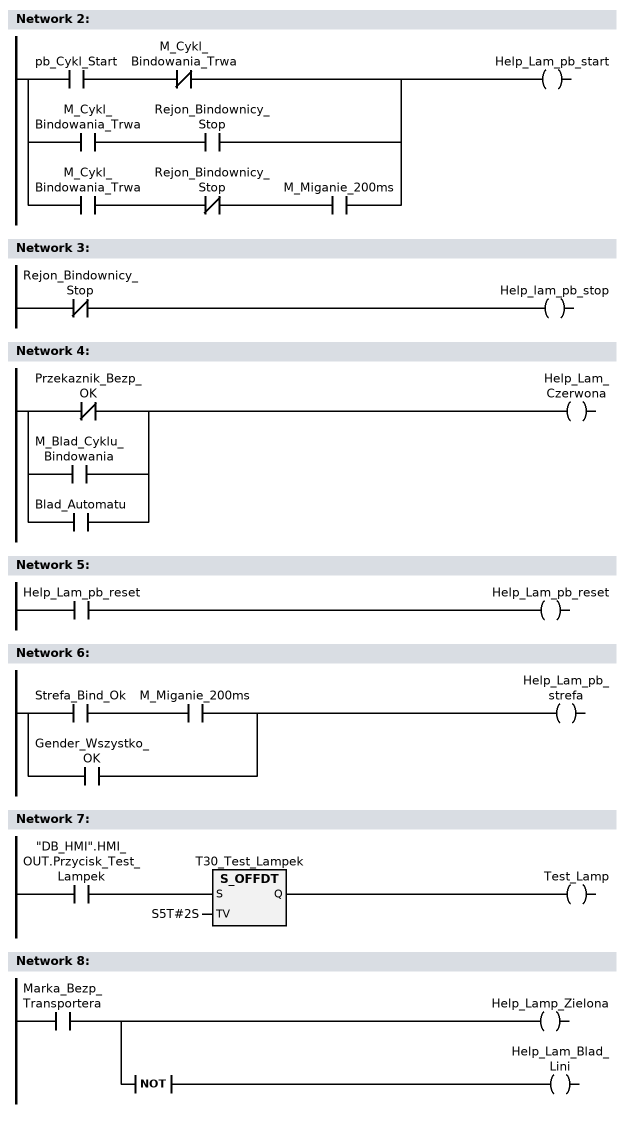
[picture p141: Sterwanie_Swiatlo networks 2-8]
NETWORK
TITLE =
//Lampka pb start cyklu
      A     "pb_Cykl_Start";
      AN    "M_Cykl_Bindowania_Trwa";
      O;
      A     "M_Cykl_Bindowania_Trwa";
      A     "Rejon_Bindownicy_Stop";
      O;
      A     "M_Cykl_Bindowania_Trwa";
      AN    "Rejon_Bindownicy_Stop";
      A     "M_Miganie_200ms";
      =     "Help_Lam_pb_start";
NETWORK
TITLE =
//Lampka stop
      AN    "Rejon_Bindownicy_Stop";
      =     "Help_lam_pb_stop";
NETWORK
TITLE =
      ON    "Przekaznik_Bezp_OK";
      O     "M_Blad_Cyklu_Bindowania";
      O     "Blad_Automatu";
      =     "Help_Lam_Czerwona";
NETWORK
TITLE =
//Miga reset
      A     "Help_Lam_pb_reset";
      =     "Help_Lam_pb_reset";
NETWORK
TITLE =
//Lampka bezpieczenstwa strefa
      A     "Strefa_Bind_Ok";
      A     "M_Miganie_200ms";
      O     "Gender_Wszystko_OK";
      =     "Help_Lam_pb_strefa";
NETWORK
TITLE =
//Test Lampek z timmerem przedluzonym
      A     "DB_HMI".HMI_OUT.Przycisk_Test_Lampek;
      L     S5T#2S;
      SF    "T30_Test_Lampek";
      NOP   0;
      NOP   0;
      NOP   0;
      A     "T30_Test_Lampek";
      =     "Test_Lamp";
NETWORK
TITLE =
//linia pracuje
      A     "Marka_Bezp_Transportera";
      =     L 1.0;
      A     L 1.0;
      BLD   102;
      =     "Help_Lamp_Zielona";
      A     L 1.0;
      NOT;
      =     "Help_Lam_Blad_Lini";
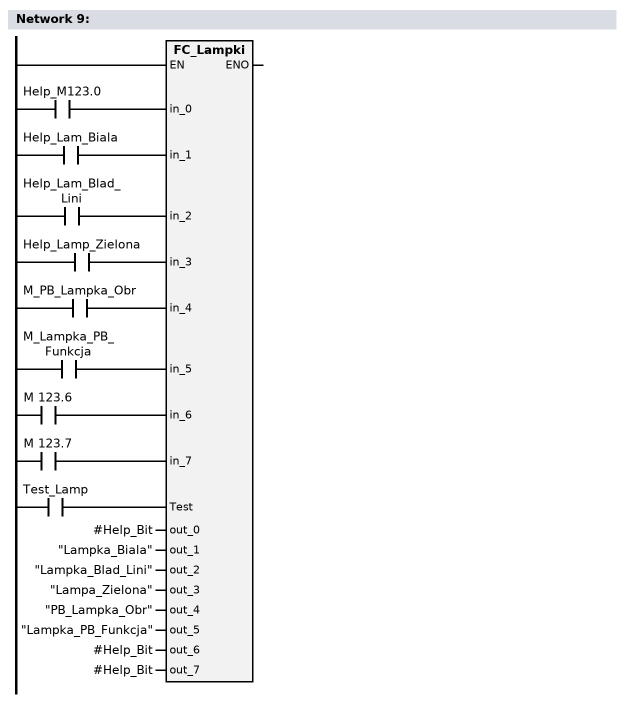
NETWORK
TITLE =
//Lampki na szafie sterowniczej sa troche przesuniete bo brakuje zielonej
      A     "Help_M123.0";
      =     L 1.0;
      BLD   103;
      A     "Help_Lam_Biala";
      =     L 1.1;
      BLD   103;
      A     "Help_Lam_Blad_Lini";
      =     L 1.2;
      BLD   103;
      A     "Help_Lamp_Zielona";
      =     L 1.3;
      BLD   103;
      A     "M_PB_Lampka_Obr";
      =     L 1.4;
      BLD   103;
      A     "M_Lampka_PB_Funkcja";
      =     L 1.5;
      BLD   103;
      A     M 123.6;
      =     L 1.6;
      BLD   103;
      A     M 123.7;
      =     L 1.7;
      BLD   103;
      A     "Test_Lamp";
      =     L 2.0;
      BLD   103;
      CALL  "FC_Lampki" (
           in_0                     := L 1.0,
           in_1                     := L 1.1,
           in_2                     := L 1.2,
           in_3                     := L 1.3,
           in_4                     := L 1.4,
           in_5                     := L 1.5,
           in_6                     := L 1.6,
           in_7                     := L 1.7,
           Test                     := L 2.0,
           out_0                    := #Help_Bit,
           out_1                    := "Lampka_Biala",
           out_2                    := "Lampka_Blad_Lini",
           out_3                    := "Lampa_Zielona",
           out_4                    := "PB_Lampka_Obr",
           out_5                    := "Lampka_PB_Funkcja",
           out_6                    := #Help_Bit,
           out_7                    := #Help_Bit);
      NOP   0;
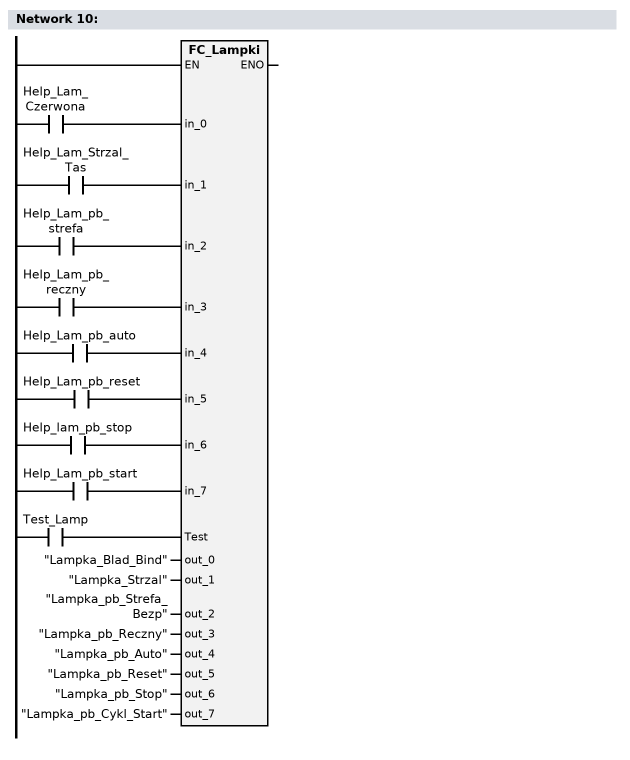
NETWORK
TITLE =
//funkcja zarzadzajaca lampami
//Lampki na panelu operatorskim
      A     "Help_Lam_Czerwona";
      =     L 1.0;
      BLD   103;
      A     "Help_Lam_Strzal_Tas";
      =     L 1.1;
      BLD   103;
      A     "Help_Lam_pb_strefa";
      =     L 1.2;
      BLD   103;
      A     "Help_Lam_pb_reczny";
      =     L 1.3;
      BLD   103;
      A     "Help_Lam_pb_auto";
      =     L 1.4;
      BLD   103;
      A     "Help_Lam_pb_reset";
      =     L 1.5;
      BLD   103;
      A     "Help_lam_pb_stop";
      =     L 1.6;
      BLD   103;
      A     "Help_Lam_pb_start";
      =     L 1.7;
      BLD   103;
      A     "Test_Lamp";
      =     L 2.0;
      BLD   103;
      CALL  "FC_Lampki" (
           in_0                     := L 1.0,
           in_1                     := L 1.1,
           in_2                     := L 1.2,
           in_3                     := L 1.3,
           in_4                     := L 1.4,
           in_5                     := L 1.5,
           in_6                     := L 1.6,
           in_7                     := L 1.7,
           Test                     := L 2.0,
           out_0                    := "Lampka_Blad_Bind",
           out_1                    := "Lampka_Strzal",
           out_2                    := "Lampka_pb_Strefa_Bezp",
           out_3                    := "Lampka_pb_Reczny",
           out_4                    := "Lampka_pb_Auto",
           out_5                    := "Lampka_pb_Reset",
           out_6                    := "Lampka_pb_Stop",
           out_7                    := "Lampka_pb_Cykl_Start");
      NOP   0;
END_FUNCTION

FUNCTION "Przyciski_Dwufunkcyjne" : VOID	// FC 11
AUTHOR : Kng
NAME : Help_FC
VERSION : 0.1
VAR_INPUT
  Kierunek_Prawo : BOOL ;
  Kierunek_Lewo : BOOL ;
  Funkcja : BOOL ;
END_VAR
VAR_OUTPUT
  Jazda_Prawo : BOOL ;
  Jazda_Lewo : BOOL ;
  Obrot_Prawo : BOOL ;
  Obrot_Lewo : BOOL ;
END_VAR
BEGIN
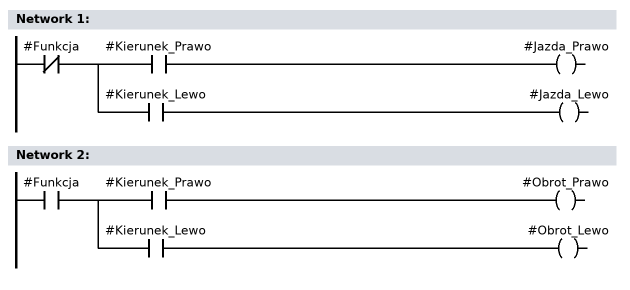
NETWORK
TITLE =
      AN    #Funkcja;
      =     L 0.0;
      A     L 0.0;
      A     #Kierunek_Prawo;
      =     #Jazda_Prawo;
      A     L 0.0;
      A     #Kierunek_Lewo;
      =     #Jazda_Lewo;
NETWORK
TITLE =
      A     #Funkcja;
      =     L 0.0;
      A     L 0.0;
      A     #Kierunek_Prawo;
      =     #Obrot_Prawo;
      A     L 0.0;
      A     #Kierunek_Lewo;
      =     #Obrot_Lewo;
END_FUNCTION

FUNCTION "Przyporzadkowanie_Wejsc" : VOID	// FC 20
//Pobranie z bloku db stanu wejsc sieci asi i przyporzadkowanie do odpowiedniego 
//urzadzenia lini.
//NW35-adresy B
//
//
//Opis sygnalow od bindownicy:
//banda 23, 24, 1, 2 tworza zestaw tasm maszyny bindujacej
//obr 15 to obrotnica bindownicy
//25,26- to kurtyny
//16-rygiel
//17-modul resetu
AUTHOR : Kng
NAME : Help_FC
VERSION : 0.1
VAR_TEMP
  Help_Bit_1 : BOOL ;
  Help_Bit_2 : BOOL ;
  Help_Word_1 : INT ;
  Help_Word_2 : INT ;
END_VAR
BEGIN
NETWORK
TITLE =
//Ten network celowo jest wolny
NETWORK
TITLE =
NETWORK
TITLE = Silnik ok
//Banda Adres 3
      A     "Asi_input_Transport".Adres_3_bit_0;
      =     "AIO".Banda_T3.Silnik_OK;
      A     "Asi_input_Transport".Adres_3_bit_1;
      =     "AIO".Banda_T3.Rezerwa_Silnik;
      A     "Asi_input_Transport".Adres_3_bit_2;
      =     "AIO".Banda_T3.Foto_1;
      A     "Asi_input_Transport".Adres_3_bit_3;
      =     "AIO".Banda_T3.Foto_2;
NETWORK
TITLE = Silnik ok
//Banda Adres 4
      A     "Asi_input_Transport".Adres_4_bit_0;
      =     "AIO".Banda_T4.Silnik_OK;
      A     "Asi_input_Transport".Adres_4_bit_1;
      =     "AIO".Banda_T4.Rezerwa_Silnik;
      A     "Asi_input_Transport".Adres_4_bit_2;
      =     "AIO".Banda_T4.Foto_1;
      A     "Asi_input_Transport".Adres_4_bit_3;
      =     "AIO".Banda_T4.Foto_2;
NETWORK
TITLE = Silnik ok
//Banda Adres 5
      A     "Asi_input_Transport".Adres_5_bit_0;
      =     "AIO".Banda_T5.Silnik_OK;
      A     "Asi_input_Transport".Adres_5_bit_1;
      =     "AIO".Banda_T5.Rezerwa_Silnik;
      A     "Asi_input_Transport".Adres_5_bit_2;
      =     "AIO".Banda_T5.Foto_1;
      A     "Asi_input_Transport".Adres_5_bit_3;
      =     "AIO".Banda_T5.Foto_2;
NETWORK
TITLE = Silnik ok
//Banda Adres 6
      A     "Asi_input_Transport".Adres_6_bit_0;
      =     "AIO".Banda_T6.Silnik_OK;
      A     "Asi_input_Transport".Adres_6_bit_1;
      =     "AIO".Banda_T6.Rezerwa_Silnik;
      A     "Asi_input_Transport".Adres_6_bit_2;
      =     "AIO".Banda_T6.Foto_1;
      A     "Asi_input_Transport".Adres_6_bit_3;
      =     "AIO".Banda_T6.Foto_2;
NETWORK
TITLE = Silnik ok
//Banda Adres 7
      A     "Asi_input_Transport".Adres_7_bit_0;
      =     "AIO".Banda_T7.Silnik_OK;
      A     "Asi_input_Transport".Adres_7_bit_1;
      =     "AIO".Banda_T7.Rezerwa_Silnik;
      A     "Asi_input_Transport".Adres_7_bit_2;
      =     "AIO".Banda_T7.Foto_1;
      A     "Asi_input_Transport".Adres_7_bit_3;
      =     "AIO".Banda_T7.Foto_2;
NETWORK
TITLE = Silnik ok
//Banda Adres 8
      A     "Asi_input_Transport".Adres_8_bit_0;
      =     "AIO".Banda_T8.Silnik_OK;
      A     "Asi_input_Transport".Adres_8_bit_1;
      =     "AIO".Banda_T8.Rezerwa_Silnik;
      A     "Asi_input_Transport".Adres_8_bit_2;
      =     "AIO".Banda_T8.Foto_1;
      A     "Asi_input_Transport".Adres_8_bit_3;
      =     "AIO".Banda_T8.Foto_2;
NETWORK
TITLE = Silnik ok
//Banda Adres 9
      A     "Asi_input_Transport".Adres_9_bit_0;
      =     "AIO".Banda_T9.Silnik_OK;
      A     "Asi_input_Transport".Adres_9_bit_1;
      =     "AIO".Banda_T9.Rezerwa_Silnik;
      A     "Asi_input_Transport".Adres_9_bit_2;
      =     "AIO".Banda_T9.Foto_1;
      A     "Asi_input_Transport".Adres_9_bit_3;
      =     "AIO".Banda_T9.Foto_2;
//Info do foliarki o zajetosci lini
      A     "AIO".Banda_T9.Foto_1;
      =     "MPI_GD".OUT.Foto_Banda_9;
//-
NETWORK
TITLE = Silnik ok
//Banda Adres 10.Banda nalezy do foliarki.
      A     "Asi_input_Transport".Adres_10_bit_0;
      =     "AIO".Banda_T10.Silnik_OK;
      A     "Asi_input_Transport".Adres_10_bit_1;
      =     "AIO".Banda_T10.Rezerwa_Silnik;
      A     "Asi_input_Transport".Adres_10_bit_2;
      =     "AIO".Banda_T10.Foto_1;
      A     "Asi_input_Transport".Adres_10_bit_3;
      =     "AIO".Banda_T10.Foto_2;
//Sygnaly do foliarki
      A     "AIO".Banda_T10.Silnik_OK;
      =     "MPI_GD".OUT.Silnik_10_OK;
//-
      A     "AIO".Banda_T10.Foto_1;
      =     "MPI_GD".OUT.Foto_1_Banda_10;
//-
      A     "AIO".Banda_T10.Foto_2;
      =     "MPI_GD".OUT.Foto_2_Banda_10;
NETWORK
TITLE = Silnik ok
//Banda Adres 11. Banda nalezy do foliarki.
      A     "Asi_input_Transport".Adres_11_bit_0;
      =     "AIO".Banda_T11.Silnik_OK;
      A     "Asi_input_Transport".Adres_11_bit_1;
      =     "AIO".Banda_T11.Rezerwa_Silnik;
      A     "Asi_input_Transport".Adres_11_bit_2;
      =     "AIO".Banda_T11.Foto_1;
      A     "Asi_input_Transport".Adres_11_bit_3;
      =     "AIO".Banda_T11.Foto_2;
//Sygnaly do foliarki
      A     "AIO".Banda_T11.Silnik_OK;
      =     "MPI_GD".OUT.Silnik_11_OK;
//-
      A     "AIO".Banda_T11.Foto_1;
      =     "MPI_GD".OUT.Foto_Banda_11;
NETWORK
TITLE = Silnik ok
//Banda Adres 12
      A     "Asi_input_Transport".Adres_12_bit_0;
      =     "AIO".Banda_T12.Silnik_OK;
      A     "Asi_input_Transport".Adres_12_bit_1;
      =     "AIO".Banda_T12.Rezerwa_Silnik;
      A     "Asi_input_Transport".Adres_12_bit_2;
      =     "AIO".Banda_T12.Foto_1;
      A     "Asi_input_Transport".Adres_12_bit_3;
      =     "AIO".Banda_T12.Foto_2;
NETWORK
TITLE = Silnik ok
//Banda Adres 13
      A     "Asi_input_Transport".Adres_13_bit_0;
      =     "AIO".Banda_T13.Silnik_OK;
      A     "Asi_input_Transport".Adres_13_bit_1;
      =     "AIO".Banda_T13.Rezerwa_Silnik;
      A     "Asi_input_Transport".Adres_13_bit_2;
      =     "AIO".Banda_T13.Foto_1;
      A     "Asi_input_Transport".Adres_13_bit_3;
      =     "AIO".Banda_T13.Foto_2;
NETWORK
TITLE = Silnik ok
//Banda Adres 14
      A     "Asi_input_Transport".Adres_14_bit_0;
      =     "AIO".Banda_T14.Silnik_OK;
      A     "Asi_input_Transport".Adres_14_bit_1;
      =     "AIO".Banda_T14.Rezerwa_Silnik;
      A     "Asi_input_Transport".Adres_14_bit_2;
      =     "AIO".Banda_T14.Foto_1;
      A     "Asi_input_Transport".Adres_14_bit_3;
      =     "AIO".Banda_T14.Foto_2;
NETWORK
TITLE = Silnik ok
//Obrotnica Adres_18 
      A     "Asi_input_Transport".Adres_18_bit_0;
      =     "AIO".Obr_T18.Silnik_OK;
      A     "Asi_input_Transport".Adres_18_bit_1;
      =     "AIO".Obr_T18.Rezerwa_Silnik;
      A     "Asi_input_Transport".Adres_18_bit_2;
      =     "AIO".Obr_T18.Foto_1;
      A     "Asi_input_Transport".Adres_18_bit_3;
      =     "AIO".Obr_T18.Foto_2;
NETWORK
TITLE = Silnik ok
//Czujniki obrotnicy 1 Adres 19
      A     "Asi_input_Transport".Adres_19_bit_0;
      =     "AIO".Czuj_T19.Czujnik_0_St;
      A     "Asi_input_Transport".Adres_19_bit_1;
      =     "AIO".Czuj_T19.Czujnik_Ham_0_St;
      A     "Asi_input_Transport".Adres_19_bit_2;
      =     "AIO".Czuj_T19.Czujnik_Ham_90_St;
      A     "Asi_input_Transport".Adres_19_bit_3;
      =     "AIO".Czuj_T19.Czujnik_90_St;
NETWORK
TITLE = Silnik ok
//Obrotnica Adres 20
      A     "Asi_input_Transport".Adres_20_bit_0;
      =     "AIO".Obr_T20.Silnik_OK;
      A     "Asi_input_Transport".Adres_20_bit_1;
      =     "AIO".Obr_T20.Rezerwa_Silnik;
      A     "Asi_input_Transport".Adres_20_bit_2;
      =     "AIO".Obr_T20.Foto_1;
      A     "Asi_input_Transport".Adres_20_bit_3;
      =     "AIO".Obr_T20.Foto_2;
NETWORK
TITLE = Silnik ok
//Czujniki Obrotnicy 2 Adres 21
      A     "Asi_input_Transport".Adres_21_bit_0;
      =     "AIO".Czuj_T21.Czujnik_0_St;
      A     "Asi_input_Transport".Adres_21_bit_1;
      =     "AIO".Czuj_T21.Czujnik_Ham_0_St;
      A     "Asi_input_Transport".Adres_21_bit_2;
      =     "AIO".Czuj_T21.Czujnik_Ham_90_St;
      A     "Asi_input_Transport".Adres_21_bit_3;
      =     "AIO".Czuj_T21.Czujnik_90_St;
NETWORK
TITLE = Silnik ok
//Czujniki Obrotnicy 2 Adres 22
      A     "Asi_input_Transport".Adres_22_bit_0;
      =     "AIO".Czuj_T22.Czujnik_45_St_CW;
      A     "Asi_input_Transport".Adres_22_bit_1;
      =     "AIO".Czuj_T22.Czujnik_45_St_CCW;
      A     "Asi_input_Transport".Adres_22_bit_2;
      =     "AIO".Czuj_T22.Rez_0_2;
      A     "Asi_input_Transport".Adres_22_bit_3;
      =     "AIO".Czuj_T22.Rez_0_3;
NETWORK
TITLE = Silnik ok
//Sprawdzenie czujnikow Bezpieczenstwa lini
//Not Aus 27 
      A     "Asi_input_Transport".Adres_27_bit_0;
      =     "AIO".ESTOP_T27.EStop_Tor_1_1;
      A     "Asi_input_Transport".Adres_27_bit_1;
      =     "AIO".ESTOP_T27.EStop_Tor_1_2;
      A     "Asi_input_Transport".Adres_27_bit_2;
      =     "AIO".ESTOP_T27.EStop_Tor_2_1;
      A     "Asi_input_Transport".Adres_27_bit_3;
      =     "AIO".ESTOP_T27.EStop_Tor_2_2;
NETWORK
TITLE =
//Sprawdzenie czujnikow Bezpieczenstwa lini
//Not Aus 28
      A     "Asi_input_Transport".Adres_28_bit_0;
      =     "AIO".ESTOP_T28.EStop_Tor_1_1;
      A     "Asi_input_Transport".Adres_28_bit_1;
      =     "AIO".ESTOP_T28.EStop_Tor_1_2;
      A     "Asi_input_Transport".Adres_28_bit_2;
      =     "AIO".ESTOP_T28.EStop_Tor_2_1;
      A     "Asi_input_Transport".Adres_28_bit_3;
      =     "AIO".ESTOP_T28.EStop_Tor_2_2;
NETWORK
TITLE =
//Sprawdzenie czujnikow Bezpieczenstwa lini
//Not Aus 29
      A     "Asi_input_Transport".Adres_29_bit_0;
      =     "AIO".ESTOP_T29.EStop_Tor_1_1;
      A     "Asi_input_Transport".Adres_29_bit_1;
      =     "AIO".ESTOP_T29.EStop_Tor_1_2;
      A     "Asi_input_Transport".Adres_29_bit_2;
      =     "AIO".ESTOP_T29.EStop_Tor_2_1;
      A     "Asi_input_Transport".Adres_29_bit_3;
      =     "AIO".ESTOP_T29.EStop_Tor_2_2;
NETWORK
TITLE =
//Sprawdzenie czujnikow Bezpieczenstwa lini
//Not Aus 30
      A     "Asi_input_Transport".Adres_30_bit_0;
      =     "AIO".ESTOP_T30.EStop_Tor_1_1;
      A     "Asi_input_Transport".Adres_30_bit_1;
      =     "AIO".ESTOP_T30.EStop_Tor_1_2;
      A     "Asi_input_Transport".Adres_30_bit_2;
      =     "AIO".ESTOP_T30.EStop_Tor_2_1;
      A     "Asi_input_Transport".Adres_30_bit_3;
      =     "AIO".ESTOP_T30.EStop_Tor_2_2;
END_FUNCTION

FUNCTION "Przyporzadkowanie_Wyjsc" : VOID	// FC 21
VERSION : 0.1
VAR_TEMP
  Temp_Word_1 : INT ;
  Help_Bit_1 : BOOL ;
END_VAR
BEGIN
NETWORK
TITLE =
//Ten Network celowo jest wolny
NETWORK
TITLE = Temporary placeholder variable
//Banda 3 Adres 3
//****************ClockWise*******************
      A     "Zawsze_False";	//C_Wise
      =     "Asi_output_Transport".Adres_3_bit_0;
//****************CounterClockWise************
      A     "AIO".Banda_T3.C_Wise;
      =     "Asi_output_Transport".Adres_3_bit_1;	//CC_Wise
//****************Wolno***********************
      A     "Zawsze_True";
      =     "Asi_output_Transport".Adres_3_bit_2;	//Wolno
//****************Bit_Bezpieczenstwa**********
      A     "Marka_Bezp_Transportera";	//Safety
      =     "Asi_output_Transport".Adres_3_bit_3;
NETWORK
TITLE = Temporary placeholder variable
//Banda 4 Obrotnica
//****************ClockWise*******************
      A     "AIO".Banda_T4.C_Wise;	//C_Wise
      =     "Asi_output_Transport".Adres_4_bit_0;
//****************CounterClockWise************
      A     "AIO".Banda_T4.CC_Wise;
      =     "Asi_output_Transport".Adres_4_bit_1;	//CC_Wise
//****************Wolno***********************
      A     "Zawsze_True";
      =     "Asi_output_Transport".Adres_4_bit_2;	//Wolno
//****************Bit_Bezpieczenstwa**********
      A     "Marka_Bezp_Transportera";	//Safety
      =     "Asi_output_Transport".Adres_4_bit_3;
NETWORK
TITLE = Temporary placeholder variable
//Banda 5 Rolki
//****************ClockWise*******************
      A     "Zawsze_False";	//C_Wise
      =     "Asi_output_Transport".Adres_5_bit_0;
//****************CounterClockWise************
      A     "AIO".Banda_T5.C_Wise;
      =     "Asi_output_Transport".Adres_5_bit_1;	//CC_Wise
//****************Wolno***********************
      A     "Zawsze_True";
      =     "Asi_output_Transport".Adres_5_bit_2;	//Wolno
//****************Bit_Bezpieczenstwa**********
      A     "Marka_Bezp_Transportera";	//Safety
      =     "Asi_output_Transport".Adres_5_bit_3;
NETWORK
TITLE = Temporary placeholder variable
//Banda 6 Rolki
//****************ClockWise*******************
      A     "AIO".Banda_T6.C_Wise;	//C_Wise
      =     "Asi_output_Transport".Adres_6_bit_0;
//****************CounterClockWise************
      A     "Zawsze_False";
      =     "Asi_output_Transport".Adres_6_bit_1;	//CC_Wise
//****************Wolno***********************
      A     "Zawsze_False";
      =     "Asi_output_Transport".Adres_6_bit_2;	//Wolno
//****************Bit_Bezpieczenstwa**********
      A     "Marka_Bezp_Transportera";	//Safety
      =     "Asi_output_Transport".Adres_6_bit_3;
NETWORK
TITLE = Temporary placeholder variable
//Banda 7 Rolki
//****************ClockWise*******************
      A     "Zawsze_False";	//C_Wise
      =     "Asi_output_Transport".Adres_7_bit_0;
//****************CounterClockWise************
      A     "AIO".Banda_T7.C_Wise;
      =     "Asi_output_Transport".Adres_7_bit_1;	//CC_Wise
//****************Wolno***********************
      A     "Zawsze_True";
      =     "Asi_output_Transport".Adres_7_bit_2;	//Wolno
//****************Bit_Bezpieczenstwa**********
      A     "Marka_Bezp_Transportera";	//Safety
      =     "Asi_output_Transport".Adres_7_bit_3;
NETWORK
TITLE = Temporary placeholder variable
//Banda 8 Rolki
//****************ClockWise*******************
      A     "AIO".Banda_T8.C_Wise;	//C_Wise
      =     "Asi_output_Transport".Adres_8_bit_0;
//****************CounterClockWise************
      A     "Zawsze_False";
      =     "Asi_output_Transport".Adres_8_bit_1;	//CC_Wise
//****************Wolno***********************
      A     "Zawsze_False";
      =     "Asi_output_Transport".Adres_8_bit_2;	//Wolno
//****************Bit_Bezpieczenstwa**********
      A     "Marka_Bezp_Transportera";	//Safety
      =     "Asi_output_Transport".Adres_8_bit_3;
NETWORK
TITLE = Temporary placeholder variable
//Banda 9 Rolki
//****************ClockWise*******************
      A     "Zawsze_False";	//C_Wise
      =     "Asi_output_Transport".Adres_9_bit_0;
//****************CounterClockWise************
      A     "AIO".Banda_T9.C_Wise;
      =     "Asi_output_Transport".Adres_9_bit_1;	//CC_Wise
//****************Wolno***********************
      A     "Zawsze_True";
      =     "Asi_output_Transport".Adres_9_bit_2;	//Wolno
//****************Bit_Bezpieczenstwa**********
      A     "Marka_Bezp_Transportera";	//Safety
      =     "Asi_output_Transport".Adres_9_bit_3;
NETWORK
TITLE = Temporary placeholder variable
//Banda 10 Rolki
//Uwaga Banda ta nalezy do foliarki
//Sygnaly z foliarki
      A     "MPI_GD".IN.Motor_10_Lewo;
      =     "AIO".Banda_T10.C_Wise;
      A     "MPI_GD".IN.Motor_10_Prawo;
      =     "AIO".Banda_T10.CC_Wise;
//****************ClockWise*******************
      A     "AIO".Banda_T10.C_Wise;	//C_Wise
      =     "Asi_output_Transport".Adres_10_bit_0;
//****************CounterClockWise************
      A     "AIO".Banda_T10.CC_Wise;
      =     "Asi_output_Transport".Adres_10_bit_1;	//CC_Wise
//****************Wolno***********************
      A     "Zawsze_True";
      =     "Asi_output_Transport".Adres_10_bit_2;	//Wolno
//****************Bit_Bezpieczenstwa**********
      A     "Marka_Bezp_Transportera";	//Safety
      =     "Asi_output_Transport".Adres_10_bit_3;
NETWORK
TITLE = Temporary placeholder variable
//Banda 11 Rolki
//Uwaga Banda ta nalezy do foliarki
//Sygnaly z foliarki
      A     "MPI_GD".IN.Motor_11_Lewo;
      =     "AIO".Banda_T11.C_Wise;
      A     "MPI_GD".IN.Motor_11_Prawo;
      =     "AIO".Banda_T11.CC_Wise;
//****************ClockWise*******************
      A     "AIO".Banda_T11.C_Wise;	//C_Wise
      =     "Asi_output_Transport".Adres_11_bit_0;
//****************CounterClockWise************
      A     "AIO".Banda_T11.CC_Wise;
      =     "Asi_output_Transport".Adres_11_bit_1;	//CC_Wise
//****************Wolno***********************
      A     "Zawsze_True";
      =     "Asi_output_Transport".Adres_11_bit_2;	//Wolno
//****************Bit_Bezpieczenstwa**********
      A     "Marka_Bezp_Transportera";	//Safety
      =     "Asi_output_Transport".Adres_11_bit_3;
NETWORK
TITLE = Temporary placeholder variable
//Banda 12 Rolki wlot 2 na obrotnice
//****************ClockWise*******************
      A     "AIO".Banda_T12.C_Wise;	//C_Wise
      =     "Asi_output_Transport".Adres_12_bit_0;
//****************CounterClockWise************
      A     "Zawsze_False";
      =     "Asi_output_Transport".Adres_12_bit_1;	//CC_Wise
//****************Wolno***********************
      A     "Zawsze_False";
      =     "Asi_output_Transport".Adres_12_bit_2;	//Wolno
//****************Bit_Bezpieczenstwa**********
      A     "Marka_Bezp_Transportera";	//Safety
      =     "Asi_output_Transport".Adres_12_bit_3;
NETWORK
TITLE = Temporary placeholder variable
//Banda 13 Adres 13 Rolki na obrotnicy
//****************ClockWise*******************
      A     "AIO".Banda_T13.C_Wise;	//C_Wise
      =     "Asi_output_Transport".Adres_13_bit_0;
//****************CounterClockWise************
      A     "AIO".Banda_T13.CC_Wise;
      =     "Asi_output_Transport".Adres_13_bit_1;	//CC_Wise
//****************Wolno***********************
      A     "Zawsze_False";
      =     "Asi_output_Transport".Adres_13_bit_2;	//Wolno
//****************Bit_Bezpieczenstwa**********
      A     "Marka_Bezp_Transportera";	//Safety
      =     "Asi_output_Transport".Adres_13_bit_3;
NETWORK
TITLE = Temporary placeholder variable
//Banda 14 Adres 14 Wylot z maszyny
//****************ClockWise*******************
      A     "AIO".Banda_T14.C_Wise;	//C_Wise
      =     "Asi_output_Transport".Adres_14_bit_0;
//****************CounterClockWise************
      A     "Zawsze_False";
      =     "Asi_output_Transport".Adres_14_bit_1;	//CC_Wise
//****************Wolno***********************
      A     "Zawsze_False";
      =     "Asi_output_Transport".Adres_14_bit_2;	//Wolno
//****************Bit_Bezpieczenstwa**********
      A     "Marka_Bezp_Transportera";	//Safety
      =     "Asi_output_Transport".Adres_14_bit_3;
NETWORK
TITLE = Temporary placeholder variable
//Obrotnica 18  Adres 18 
//****************ClockWise*******************
      A     "AIO".Obr_T18.C_Wise;
      =     "Asi_output_Transport".Adres_18_bit_0;
//****************CounterClockWise************
      A     "AIO".Obr_T18.CC_Wise;
      =     "Asi_output_Transport".Adres_18_bit_1;	//CC_Wise
//****************Wolno***********************
      A     "AIO".Obr_T18.Wolno;
      =     "Asi_output_Transport".Adres_18_bit_2;	//Wolno
//****************Bit_Bezpieczenstwa**********
      A     "Marka_Bezp_Transportera";	//Safety
      =     "Asi_output_Transport".Adres_18_bit_3;
NETWORK
TITLE = Temporary placeholder variable
//Obrotnica 20 Adres 20
//****************ClockWise*******************
      A     "AIO".Obr_T20.C_Wise;
      =     "Asi_output_Transport".Adres_20_bit_0;
//****************CounterClockWise************
      A     "AIO".Obr_T20.CC_Wise;
      =     "Asi_output_Transport".Adres_20_bit_1;	//CC_Wise
//****************Wolno***********************
      A     "AIO".Obr_T20.Wolno;
      =     "Asi_output_Transport".Adres_20_bit_2;	//Wolno
//****************Bit_Bezpieczenstwa**********
      A     "Marka_Bezp_Transportera";	//Safety
      =     "Asi_output_Transport".Adres_20_bit_3;
NETWORK
TITLE = Temporary placeholder variable
//Adres 21, 22 Brak Output
NETWORK
TITLE =
//Aedrs 27,28,29,30,31. Adresy ESTOP brak syganlow output
NETWORK
TITLE =
//Dziekuje za uwage
END_FUNCTION

FUNCTION "Przyp_Wejsc_Gender" : VOID	// FC 22
//Pobranie z bloku db stanu wejsc sieci asi i przyporzadkowanie do odpowiedniego 
//urzadzenia lini.
//NW35-adresy B
//
//
//Opis sygnalow od bindownicy:
//banda 23, 24, 1, 2 tworza zestaw tasm maszyny bindujacej
//obr 15 to obrotnica bindownicy
//25,26- to kurtyny
//16-rygiel
//17-modul resetu
AUTHOR : Kng
NAME : Help_FC
VERSION : 0.1
VAR_TEMP
  Help_Bit_1 : BOOL ;
  Help_Bit_2 : BOOL ;
  Help_Word_1 : INT ;
  Help_Word_2 : INT ;
END_VAR
BEGIN
NETWORK
TITLE =
//Ten network celowo jest wolny
NETWORK
TITLE =
NETWORK
TITLE = Silnik ok
//Banda Adres 1 (nowy) rolki obrotnica
      A     "Asi_Input_Gender".Adres_1_bit_0;
      O     "Zawsze_True";	//dodane
      =     "AIO".Banda_G1.Silnik_OK;
      A     "Asi_Input_Gender".Adres_1_bit_1;
      =     "AIO".Banda_G1.Rezerwa_Silnik;
      A     "Asi_Input_Gender".Adres_1_bit_2;
      =     "AIO".Banda_G1.Foto_1;
      A     "Asi_Input_Gender".Adres_1_bit_3;
      =     "AIO".Banda_G1.Foto_2;
NETWORK
TITLE = Silnik ok
//Banda Adres 2 (nowy)
      A     "Asi_Input_Gender".Adres_2_bit_0;
      O     "Zawsze_True";
      =     "AIO".Banda_G2.Silnik_OK;
      A     "Asi_Input_Gender".Adres_2_bit_1;
      =     "AIO".Banda_G2.Rezerwa_Silnik;
      A     "Asi_Input_Gender".Adres_2_bit_2;
      =     "AIO".Banda_G2.Foto_1;
      A     "Asi_Input_Gender".Adres_2_bit_3;
      =     "AIO".Banda_G2.Foto_2;
NETWORK
TITLE = Silnik ok
//Obrotnica Adres 15 (nowy)
      A     "Asi_Input_Gender".Adres_15_bit_0;
      =     "AIO".Obr_G15.Silnik_OK;
      A     "Asi_Input_Gender".Adres_15_bit_1;
      =     "AIO".Obr_G15.Rezerwa_Silnik;
      A     "Asi_Input_Gender".Adres_15_bit_2;
      =     "AIO".Obr_G15.Foto_1;
      A     "Asi_Input_Gender".Adres_15_bit_3;
      =     "AIO".Obr_G15.Foto_2;
NETWORK
TITLE = Silnik ok
//Uwaga modul safety !!! (nowy)
//Rygiel Adres 16
      A     "Asi_Input_Gender".Adres_16_bit_0;
      =     "AIO".Rygiel_TG16.OSSD_Tor_1_1;
      A     "Asi_Input_Gender".Adres_16_bit_1;
      =     "AIO".Rygiel_TG16.OSSD_Tor_1_2;
      A     "Asi_Input_Gender".Adres_16_bit_2;
      =     "AIO".Rygiel_TG16.OSSD_Tor_2_1;
      A     "Asi_Input_Gender".Adres_16_bit_3;
      =     "AIO".Rygiel_TG16.OSSD_Tor_2_2;
NETWORK
TITLE = Silnik ok
//Reset kurtyn bezpieczenswa Adres 17 (nowy)
//Nie wykorzystywane wejscia
NETWORK
TITLE = Wejscie SEW 1
//Banda 23 znajdujaca sie bedaca banda wjazdowa do bindownicy (nowy)
      A     "Asi_Input_Gender".Adres_23_bit_0;
      =     "AIO".Banda_G23.Silnik_OK;
      A     "Asi_Input_Gender".Adres_23_bit_1;
      =     "AIO".Banda_G23.Rezerwa_Silnik;
      A     "Asi_Input_Gender".Adres_23_bit_2;
      =     "AIO".Banda_G23.Foto_1;
      A     "Asi_Input_Gender".Adres_23_bit_3;
      =     "AIO".Banda_G23.Foto_2;
NETWORK
TITLE = Silnik ok
//Banda 24 (nowy)
      A     "Asi_Input_Gender".Adres_24_bit_0;
      =     "AIO".Banda_G24.Silnik_OK;
      A     "Asi_Input_Gender".Adres_24_bit_1;
      =     "AIO".Banda_G24.Rezerwa_Silnik;
      A     "Asi_Input_Gender".Adres_24_bit_2;
      =     "AIO".Banda_G24.Foto_1;
      A     "Asi_Input_Gender".Adres_24_bit_3;
      =     "AIO".Banda_G24.Foto_2;
NETWORK
TITLE =
//Sprawdzenie czujnikow Bezpieczenstwa lini
//Kurtyna 25 (nowy)
      A     "Asi_Input_Gender".Adres_25_bit_0;
      =     "AIO".Kurtyna_G25.OSSD_Tor_1_1;
      A     "Asi_Input_Gender".Adres_25_bit_1;
      =     "AIO".Kurtyna_G25.OSSD_Tor_1_2;
      A     "Asi_Input_Gender".Adres_25_bit_2;
      =     "AIO".Kurtyna_G25.OSSD_Tor_2_1;
      A     "Asi_Input_Gender".Adres_25_bit_3;
      =     "AIO".Kurtyna_G25.OSSD_Tor_2_2;
NETWORK
TITLE =
//Sprawdzenie czujnikow Bezpieczenstwa lini
//Kurtyna 26 (nowy)
      A     "Asi_Input_Gender".Adres_26_bit_0;
      =     "AIO".Kurtyna_G26.OSSD_Tor_1_1;
      A     "Asi_Input_Gender".Adres_26_bit_1;
      =     "AIO".Kurtyna_G26.OSSD_Tor_1_2;
      A     "Asi_Input_Gender".Adres_26_bit_2;
      =     "AIO".Kurtyna_G26.OSSD_Tor_2_1;
      A     "Asi_Input_Gender".Adres_26_bit_3;
      =     "AIO".Kurtyna_G26.OSSD_Tor_2_2;
NETWORK
TITLE =
//Sprawdzenie czujnikow Bezpieczenstwa lini
//Not Aus 31 (nowy)
      A     "Asi_Input_Gender".Adres_31_bit_0;
      =     "AIO".ESTOP_TG31.EStop_Tor_1_1;
      A     "Asi_Input_Gender".Adres_31_bit_1;
      =     "AIO".ESTOP_TG31.EStop_Tor_1_2;
      A     "Asi_Input_Gender".Adres_31_bit_2;
      =     "AIO".ESTOP_TG31.EStop_Tor_2_1;
      A     "Asi_Input_Gender".Adres_31_bit_3;
      =     "AIO".ESTOP_TG31.EStop_Tor_2_2;
NETWORK
TITLE =
//Segment adresow B
//Dotyczy jedynie bialych modulow inuput nie zawartych wyzej
NETWORK
TITLE =
//Czujnik bindownicy Adres 19B (nowy)
      A     "Asi_Input_Gender".B_Adres_19_bit_0;
      =     "AIO".Czuj_G19_B.Czujnik_0_St;
      A     "Asi_Input_Gender".B_Adres_19_bit_1;
      =     "AIO".Czuj_G19_B.Czujnik_Ham_0_St;
      A     "Asi_Input_Gender".B_Adres_19_bit_2;
      =     "AIO".Czuj_G19_B.Czujnik_Ham_90_St;
      A     "Asi_Input_Gender".B_Adres_19_bit_3;
      =     "AIO".Czuj_G19_B.Czujnik_90_St;
NETWORK
TITLE =
//Czujnik bindownicy Adres 17B (nowy)
      A     "Asi_Input_Gender".B_Adres_17_bit_0;
      =     "AIO".Czuj_G17_B.Czujnik_Ham_180_St;
      A     "Asi_Input_Gender".B_Adres_17_bit_1;
      =     "AIO".Czuj_G17_B.Czujnik_180_St;
      A     "Asi_Input_Gender".B_Adres_17_bit_2;
      =     "AIO".Czuj_G17_B.Czujnik_Ham_270_St;
      A     "Asi_Input_Gender".B_Adres_17_bit_3;
      =     "AIO".Czuj_G17_B.Czujnik_270_St;
END_FUNCTION

FUNCTION "Przyp_Wysc_Gender" : VOID	// FC 23
VERSION : 0.1
VAR_TEMP
  Temp_Word_1 : INT ;
  Help_Bit_1 : BOOL ;
END_VAR
BEGIN
NETWORK
TITLE =
//Ten Network celowo jest wolny
NETWORK
TITLE = Temporary placeholder variable
//Banda 1 Adres 1 (nowy)
//****************ClockWise*******************
      A     "AIO".Banda_G1.CC_Wise;	//C_Wise
      =     "Asi_Output_Gender".Adres_1_bit_0;
//****************CounterClockWise************
      A     "AIO".Banda_G1.C_Wise;
      =     "Asi_Output_Gender".Adres_1_bit_1;	//CC_Wise
//****************Wolno***********************
      A     "AIO".Banda_G1.Wolno;
      O     "pb_Strefa_bezpieczenstwa";
      =     "Asi_Output_Gender".Adres_1_bit_2;	//Wolno
//****************Bit_Bezpieczenstwa**********
      A     "Marka_Bezp_Gendera";	//Safety
      =     "Asi_Output_Gender".Adres_1_bit_3;
NETWORK
TITLE = Temporary placeholder variable
//Banda 2 Adres 2 (nowy)
//****************ClockWise*******************
      A     "AIO".Banda_G2.CC_Wise;	//C_Wise
      =     "Asi_Output_Gender".Adres_2_bit_0;
//****************CounterClockWise************
      A     "AIO".Banda_G2.C_Wise;
      =     "Asi_Output_Gender".Adres_2_bit_1;	//CC_Wise
//****************Wolno***********************
      AN    "AIO".Banda_G2.Wolno;
      =     "Asi_Output_Gender".Adres_2_bit_2;	//Wolno
//****************Bit_Bezpieczenstwa**********
      A     "Marka_Bezp_Gendera";	//Safety
      =     "Asi_Output_Gender".Adres_2_bit_3;
NETWORK
TITLE = Temporary placeholder variable
//Obrotnica 15 Adres 15 (nowy)
//****************ClockWise*******************
      A     "AIO".Obr_G15.C_Wise;
      =     "Asi_Output_Gender".Adres_15_bit_0;
//****************CounterClockWise************
      A     "AIO".Obr_G15.CC_Wise;
      =     "Asi_Output_Gender".Adres_15_bit_1;	//CC_Wise
//****************Wolno***********************
      AN    "AIO".Obr_G15.Wolno;
      =     "Asi_Output_Gender".Adres_15_bit_2;	//Wolno
//****************Bit_Bezpieczenstwa**********
      A     "Marka_Bezp_Gendera";	//Safety
      =     "Asi_Output_Gender".Adres_15_bit_3;
NETWORK
TITLE =
//adres 16 rygiel brak output (nowy)
NETWORK
TITLE = Temporary placeholder variable
//adres 17 reset kurtyn (nowy)
//****************Reset wlot *****************
      A     "AIO".Reset_TG17.Reset_Wlot;
      =     "Asi_Output_Gender".Adres_17_bit_0;	//reset wlot
//****************Reset wylot ****************
      A     "AIO".Reset_TG17.Reset_Wylot;
      =     "Asi_Output_Gender".Adres_17_bit_1;	//reset wylot
NETWORK
TITLE = Temporary placeholder variable
//Banda 23 (nowy)
//
//****************ClockWise*******************
      A     "AIO".Banda_G23.CC_Wise;	//C_Wise
      =     "Asi_Output_Gender".Adres_23_bit_0;
//****************CounterClockWise************
      A     "AIO".Banda_G23.C_Wise;
      =     "Asi_Output_Gender".Adres_23_bit_1;	//CC_Wise
//****************Wolno***********************
      A     "AIO".Banda_G23.Wolno;
      =     "Asi_Output_Gender".Adres_23_bit_2;	//Wolno
//****************Bit_Bezpieczenstwa**********
      A     "Marka_Bezp_Gendera";	//Safety
      =     "Asi_Output_Gender".Adres_23_bit_3;
NETWORK
TITLE = Temporary placeholder variable
//Banda 24 (nowy)
//
//****************ClockWise*******************
      A     "AIO".Banda_G24.CC_Wise;	//C_Wise
      =     "Asi_Output_Gender".Adres_24_bit_0;
//****************CounterClockWise************
      A     "AIO".Banda_G24.C_Wise;
      =     "Asi_Output_Gender".Adres_24_bit_1;	//CC_Wise
//****************Wolno***********************
      A     "Zawsze_True";
      =     "Asi_Output_Gender".Adres_24_bit_2;	//Wolno
//****************Bit_Bezpieczenstwa**********
      A     "Marka_Bezp_Gendera";	//Safety
      =     "Asi_Output_Gender".Adres_24_bit_3;
NETWORK
TITLE =
//25,26 to kurtyny bezpieczenstwa brak output
NETWORK
TITLE =
//Aedrs 27,28,29,30,31. Adresy ESTOP brak syganlow output
NETWORK
TITLE =
//Dziekuje za uwage
END_FUNCTION

FUNCTION "Rejestr_Tasm" : VOID	// FC 30
VERSION : 0.1
BEGIN
NETWORK
TITLE =
//marki uzywane od mb60. 
//Palety sa przekazywane za pomoca rejstru przesuwnego bitowego
//Poczatek monitorowania
      O     "AIO".Banda_T4.Foto_1;
      O     "AIO".Banda_T4.Foto_2;
      A     "AIO".Banda_T4.Potw_Dost_Wlot_2;
      S     M 60.0;
//Przekazanie na pierwsza bande (banda 5)
      A     "AIO".Banda_T5.Foto_1;
      A     "AIO".Banda_T5.Paleta_Dost_do_Pop;
      A     M 60.0;
      JCN   et_1;
      S     M 60.1;
      R     M 60.0;
et_1: NOP   0;
      A     "AIO".Banda_T6.Foto_1;
      A     "AIO".Banda_T6.Paleta_Dost_do_Pop;
      A     M 60.1;
      JCN   et_2;
      S     M 60.2;
      R     M 60.1;
et_2: NOP   0;
      A     "AIO".Banda_T7.Foto_1;
      A     "AIO".Banda_T7.Paleta_Dost_do_Pop;
      A     M 60.2;
      JCN   et_3;
      S     M 60.3;
      R     M 60.2;
et_3: NOP   0;
      A     "AIO".Banda_T8.Foto_1;
      A     "AIO".Banda_T8.Paleta_Dost_do_Pop;
      A     M 60.3;
      JCN   et_4;
      S     M 60.4;
      R     M 60.3;
et_4: NOP   0;
      A     "AIO".Banda_T9.Foto_1;
      A     "AIO".Banda_T9.Paleta_Dost_do_Pop;
      A     M 60.4;
      JCN   et_5;
      S     M 60.5;
      R     M 60.4;
et_5: NOP   0;
//Banda 10 to foliarka
      A     "AIO".Banda_T10.Foto_1;
      A     "AIO".Banda_T10.Paleta_Dost_do_Pop;
      A     M 60.5;
      JCN   et_6;
      S     M 60.6;
      R     M 60.5;
et_6: NOP   0;
      A     M 60.6;
      A     "MPI_GD".IN.Foto_Banda_1;	// run in 
      S     M 62.0;
      A     M 62.0;
      A     "MPI_GD".IN.Foto_Owijarka;	//foto banda 4
      JCN   et_7;
      S     M 66.7;
      R     M 66.6;
      R     M 66.2;
et_7: NOP   0;
      A     M 66.7;
      =     "MPI_GD".OUT.Zmien_Program_Na_4;
      A     "MPI_GD".IN.Rezerwa_1;
      R     M 66.7;
//nie gotowe wiec wszystkie foliowane
      SET;
      R     "MPI_GD".OUT.Zmien_Program_Na_4;
      R     "MPI_GD".OUT.Zmien_Pragram_Na_3;
END_FUNCTION

FUNCTION "FC_Auto_Reczny" : VOID	// FC 40
//Funkcja przelaczajaca miedzy auto i recznym
VERSION : 0.1
VAR_INPUT
  Enable : BOOL ;	//Zezwolenie na dzia³anie
  Reczny : BOOL ;
  Auto : BOOL ;
  Strefa_Bezp : BOOL ;
  Test_Lampek : BOOL ;	//test lampek
  Stop : BOOL ;
  Reset_1 : BOOL ;
  Reset_2 : BOOL ;
  Reset_3 : BOOL ;
END_VAR
VAR_OUTPUT
  Lampka_Reczny : BOOL ;
  Lampka_Auto : BOOL ;
END_VAR
VAR_IN_OUT
  Auto_Reczny : BOOL ;	//Auto 1, Reczny 0
END_VAR
BEGIN
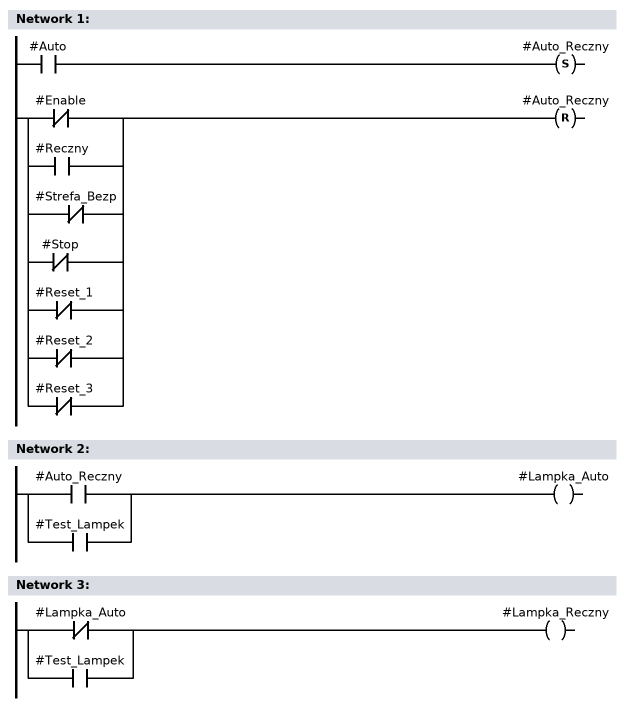
NETWORK
TITLE =
      A     #Auto;
      S     #Auto_Reczny;
      A(;
      ON    #Enable;
      O     #Reczny;
      ON    #Strefa_Bezp;
      ON    #Stop;
      ON    #Reset_1;
      ON    #Reset_2;
      ON    #Reset_3;
      );
      R     #Auto_Reczny;
      NOP   0;
NETWORK
TITLE =
      O     #Auto_Reczny;
      O     #Test_Lampek;
      =     #Lampka_Auto;
NETWORK
TITLE =
      ON    #Lampka_Auto;
      O     #Test_Lampek;
      =     #Lampka_Reczny;
END_FUNCTION

FUNCTION "Przycisk_Reset" : VOID	// FC 41
//Funkcja sluzy do jednoczesnej oblugi bledow oraz kasowania aktualnego kroku. 
//-Jezeli wcisnie sie przycisk to krotko do 5s to nastopi pruba kasowania bledu.
//-Jezeli wcisnie sie przycisk dlugo powyzej 5s to nastapi szybkie migniecie i 
//reset krokow
//
VERSION : 0.1
VAR_INPUT
  i_PB_Reset : BOOL ;
  i_T1 : TIMER ;	//Timer do dlugiego resetowania
  i_Czas_Trzymania : S5TIME ;
  i_T2 : TIMER ;	//Timer migania po przycisku
  i_Stop_Maszyny : BOOL ;
  i_Czas_Potw_Reset : S5TIME ;
  i_Clock : BOOL ;	//Zegar 100ms
END_VAR
VAR_OUTPUT
  o_Lampka_Reset : BOOL ;
END_VAR
VAR_IN_OUT
  o_Reset_Bledu : BOOL ;
  o_Reset_Krokow : BOOL ;
  io_Blok : BOOL ;
END_VAR
VAR_TEMP
  Temp_Help_1 : BOOL ;
  Temp_Help_2 : BOOL ;
END_VAR
BEGIN
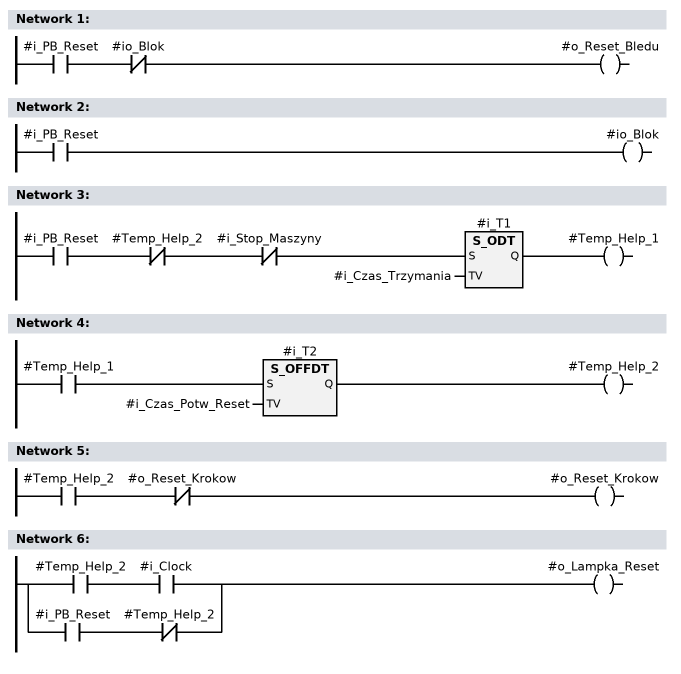
NETWORK
TITLE =
      A     #i_PB_Reset;
      AN    #io_Blok;
      =     #o_Reset_Bledu;
NETWORK
TITLE =
      A     #i_PB_Reset;
      =     #io_Blok;
NETWORK
TITLE =
      A     #i_PB_Reset;
      AN    #Temp_Help_2;
      AN    #i_Stop_Maszyny;
      L     #i_Czas_Trzymania;
      SD    #i_T1;
      NOP   0;
      NOP   0;
      NOP   0;
      A     #i_T1;
      =     #Temp_Help_1;
NETWORK
TITLE =
      A     #Temp_Help_1;
      L     #i_Czas_Potw_Reset;
      SF    #i_T2;
      NOP   0;
      NOP   0;
      NOP   0;
      A     #i_T2;
      =     #Temp_Help_2;
NETWORK
TITLE =
//Reset krokow
      A     #Temp_Help_2;
      AN    #o_Reset_Krokow;
      =     #o_Reset_Krokow;
NETWORK
TITLE =
//Lampka reset
      A     #Temp_Help_2;
      A     #i_Clock;
      O;
      A     #i_PB_Reset;
      AN    #Temp_Help_2;
      =     #o_Lampka_Reset;
END_FUNCTION

FUNCTION "ASI_Odczyt" : VOID	// FC 80
//Pobieranie danych z modulu ASI CP 342-2
AUTHOR : Kng
FAMILY : Asi_fun
NAME : r_ASi
VERSION : 0.1
VAR_INPUT
  CP_Adr : INT ;
  DB_Nr : INT ;
END_VAR
VAR_TEMP
  L_CP_Adr : DWORD ;
  L_DB_Target : WORD ;
  L_Start_Adr : DWORD ;
  L_Count : WORD ;
  Word_CP_Adr : WORD ;
  Fault : INT ;
  Target : ANY ;
END_VAR
BEGIN
NETWORK
TITLE =
      L     #CP_Adr;	// Adres urzadzenia
      SLD   3;	//Przejscie na wskaznik
      T     #L_CP_Adr;
      L     #DB_Nr;	// Nr bloku db
      T     #L_DB_Target;
      L     0;	// Start adres db 
      SLD   3;	// Przejscie na wskaznik
      T     #L_Start_Adr;
      L     4;	// Liczba petli (pobranie 16 bajtow)
next: T     #L_Count;
      L     PID [#L_CP_Adr];	// Zaladowanie wejsc
      OPN   DB [#L_DB_Target];	// Otwarcie db
      T     DBD [#L_Start_Adr];	// Wgranie danych
      L     #L_CP_Adr;	// Zaladuj adres cp
      SRD   3;	// przejscie na format obliczen
      L     4;
      +I;	// bo doble word 
      SLD   3;	// Przejscie na wskaznik
      T     #L_CP_Adr;
      L     #L_Start_Adr;	// Przesuniecie bloku danych
      SRD   3;	// do nastepnego ladowania
      L     4;
      +I;	// 
      SLD   3;	// 
      T     #L_Start_Adr;
      L     #L_Count;
      LOOP  next;	// powrot petli  next
NETWORK
TITLE =
//Recnum nie wiem co to jest dana z kart katologowych
//Funkcja ta odpowiada za segment adresowania B
      LAR1  P##Target;	// wskaznik do obszaru  docelowego
      L     W#16#1002;	//zaladuj skladnie 10 i typ byte 02
      T     LW [AR1,P#0.0];
      L     16;	//zaladuj dl. obszaru do kopiowania
      T     LW [AR1,P#2.0];
      L     #DB_Nr;	//zaladuj nr bloku db (np.:db33)
      T     LW [AR1,P#4.0];
      L     16;	//zaladuj start_adres odbioru danych
      SLD   3;	// przesun w lewo (bit ostatni ma 0.0
      OD    DW#16#84000000;	//ustaw wartosc 84-db
      T     LD [AR1,P#6.0];
//------------------------------------
      L     #CP_Adr;
      T     #Word_CP_Adr;
      CALL  "RD_REC" (
           REQ                      := TRUE,
           IOID                     := B#16#54,
           LADDR                    := #Word_CP_Adr,
           RECNUM                   := B#16#96,
           RET_VAL                  := #Fault,
           BUSY                     := L 16.1,
           RECORD                   := #Target);
END_FUNCTION

FUNCTION "ASI_Zapis" : VOID	// FC 81
//Wgranie danych do modulu ASI CP 342-2
//Funkcja ta powinna znalezc sie po programie przypiania wyjsc!!!!
AUTHOR : Kng
FAMILY : Asi_fun
NAME : w_ASi
VERSION : 0.1
VAR_INPUT
  CP_Adr : INT ;	//Adres modulu cp343-2
  DB_Nr : INT ;	//Nr db z ktorego pobierane dane
END_VAR
VAR_TEMP
  L_CP_Adr : DWORD ;
  L_DB_Target : WORD ;
  L_Start_Adr : DWORD ;
  L_Count : WORD ;
  Word_CP_Adr : WORD ;
  Fault : INT ;
  Source : ANY ;
END_VAR
BEGIN
NETWORK
TITLE =
      L     #CP_Adr;	// Adres urzadzenia
      SLD   3;	//Przejscie na wskaznik
      T     #L_CP_Adr;
      L     #DB_Nr;	// Nr bloku db
      T     #L_DB_Target;
      L     0;	// Start adres db 
      SLD   3;	// Przejscie na wskaznik
      T     #L_Start_Adr;
      L     4;	// Liczba petli (pobranie 16 bajtow)
next: T     #L_Count;
      OPN   DB [#L_DB_Target];	// Otwarcie db
      L     DBD [#L_Start_Adr];	// Zaladowanie danych
      T     PQD [#L_CP_Adr];	// Wgranie wyjsc
      L     #L_CP_Adr;	// Zaladuj adres cp
      SRD   3;	// przejscie na format obliczen
      L     4;
      +I;	// bo double word 
      SLD   3;	// Przejscie na wskaznik
      T     #L_CP_Adr;
      L     #L_Start_Adr;	// Przesuniecie bloku danych
      SRD   3;	// do nastepnego ladowania
      L     4;
      +I;	// 
      SLD   3;	// 
      T     #L_Start_Adr;
      L     #L_Count;
      LOOP  next;	// powrot petli  next
//mala maszyna to dodac beu
NETWORK
TITLE =
//Recnum nie wiem co to jest dana z kart katologowych
//Funkcja ta odpowiada za segment adresowania B
      LAR1  P##Source;	// wskaznik do obszaru  pobierajacego
      L     W#16#1002;	//zaladuj skladnie 10 i typ byte 02
      T     LW [AR1,P#0.0];
      L     16;	//zaladuj dl. obszaru do kopiowania
      T     LW [AR1,P#2.0];
      L     #DB_Nr;	//zaladuj nr bloku db (np.:db33)
      T     LW [AR1,P#4.0];
      L     16;	//zaladuj start_adres odbioru danych
      SLD   3;	// przesun w lewo (bit ostatni ma 0.0
      OD    DW#16#84000000;	//ustaw wartosc 84-db
      T     LD [AR1,P#6.0];
//------------------------------------
      L     #CP_Adr;
      T     #Word_CP_Adr;
      CALL  "WR_REC" (
           REQ                      := TRUE,
           IOID                     := B#16#55,
           LADDR                    := #Word_CP_Adr,
           RECNUM                   := B#16#96,
           RECORD                   := #Source,
           RET_VAL                  := #Fault,
           BUSY                     := L 16.1);
END_FUNCTION

FUNCTION "Opoznienie_Wylotu" : VOID	// FC 85
VERSION : 0.1
VAR_INPUT
  Wejscie : BOOL ;	//Fotokomorka
  Timmer_1 : TIMER ;
  Timmer_2 : TIMER ;
END_VAR
VAR_OUTPUT
  Wyjscie : BOOL ;
END_VAR
VAR_IN_OUT
  Zmienna : BOOL ;
END_VAR
BEGIN
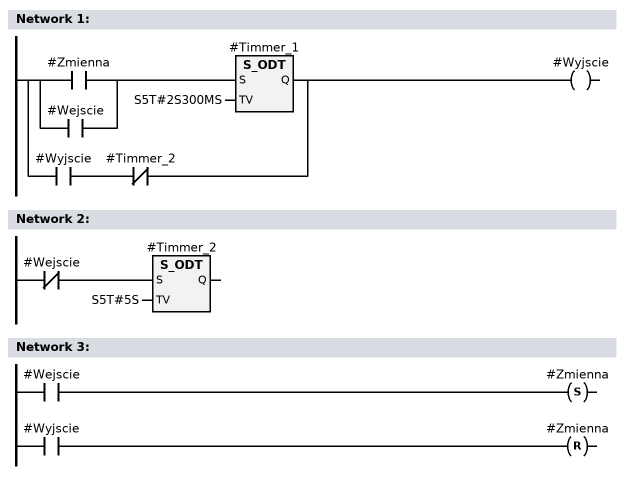
NETWORK
TITLE =
      O(;
      A(;
      O     #Zmienna;
      O     #Wejscie;
      );
      L     S5T#2S300MS;
      SD    #Timmer_1;
      NOP   0;
      NOP   0;
      NOP   0;
      A     #Timmer_1;
      );
      O;
      A     #Wyjscie;
      AN    #Timmer_2;
      =     #Wyjscie;
NETWORK
TITLE =
      AN    #Wejscie;
      L     S5T#5S;
      SD    #Timmer_2;
      NOP   0;
      NOP   0;
      NOP   0;
      NOP   0;
NETWORK
TITLE =
      A     #Wejscie;
      S     #Zmienna;
      A     #Wyjscie;
      R     #Zmienna;
      NOP   0;
END_FUNCTION

FUNCTION "Opoznienie_Wlotu" : VOID	// FC 86
VERSION : 0.1
VAR_INPUT
  Wejscie : BOOL ;	//Fotokomorka
  Timmer_1 : TIMER ;
  Timmer_2 : TIMER ;
END_VAR
VAR_OUTPUT
  Wyjscie : BOOL ;
END_VAR
VAR_IN_OUT
  Zmienna : BOOL ;
END_VAR
BEGIN
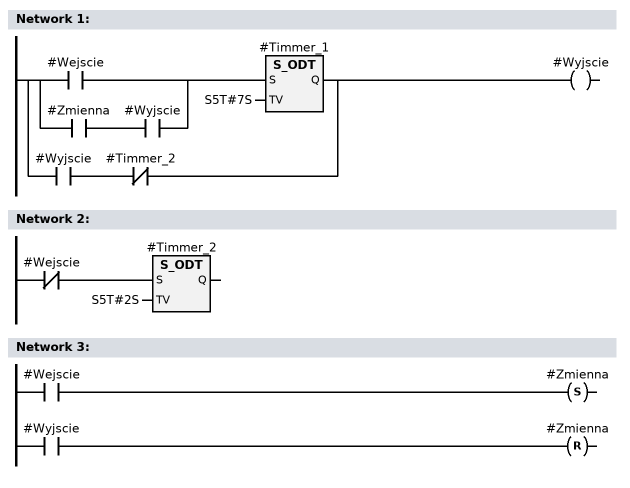
NETWORK
TITLE =
//Obecnosc palety jest aktywowana po 30s 
      O(;
      A(;
      O     #Wejscie;
      O;
      A     #Zmienna;
      A     #Wyjscie;
      );
      L     S5T#7S;
      SD    #Timmer_1;
      NOP   0;
      NOP   0;
      NOP   0;
      A     #Timmer_1;
      );
      O;
      A     #Wyjscie;
      AN    #Timmer_2;
      =     #Wyjscie;
NETWORK
TITLE =
//Filter 2s na fotokomorke aby nie zgasla gdy paleta jest na bandzie
      AN    #Wejscie;
      L     S5T#2S;
      SD    #Timmer_2;
      NOP   0;
      NOP   0;
      NOP   0;
      NOP   0;
NETWORK
TITLE =
      A     #Wejscie;
      S     #Zmienna;
      A     #Wyjscie;
      R     #Zmienna;
      NOP   0;
END_FUNCTION

FUNCTION "Komunikacja_GD" : VOID	// FC 100
VERSION : 0.1
BEGIN
NETWORK
TITLE =
//Ten network celowo jest wolny
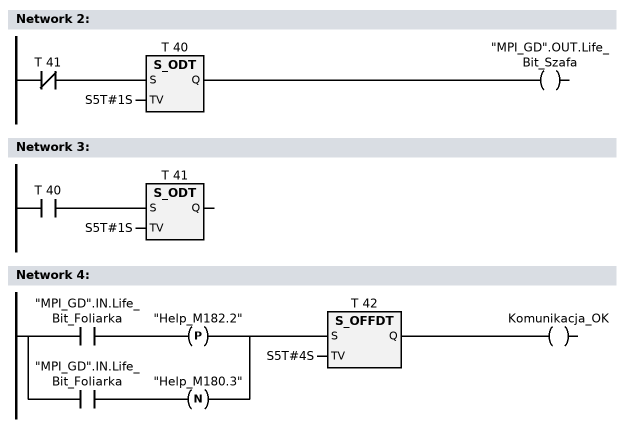
NETWORK
TITLE =
//Generator bit zycia foliarki
      AN    T 41;
      L     S5T#1S;
      SD    T 40;
      NOP   0;
      NOP   0;
      NOP   0;
      A     T 40;
      =     "MPI_GD".OUT.Life_Bit_Szafa;
NETWORK
TITLE =
//Generator bit zycia foliarki
      A     T 40;
      L     S5T#1S;
      SD    T 41;
      NOP   0;
      NOP   0;
      NOP   0;
      NOP   0;
NETWORK
TITLE =
//Sprawdzenie komunikacji z szafa transportera
      A(;
      A     "MPI_GD".IN.Life_Bit_Foliarka;
      FP    "Help_M182.2";
      O(;
      A     "MPI_GD".IN.Life_Bit_Foliarka;
      FN    "Help_M180.3";
      );
      );
      L     S5T#4S;
      SF    T 42;
      NOP   0;
      NOP   0;
      NOP   0;
      A     T 42;
      =     "Komunikacja_OK";
END_FUNCTION

FUNCTION "Obsluga bledow" : VOID	// FC 119
VERSION : 0.1
BEGIN
NETWORK
TITLE =
//Ten network celowo jest wolny
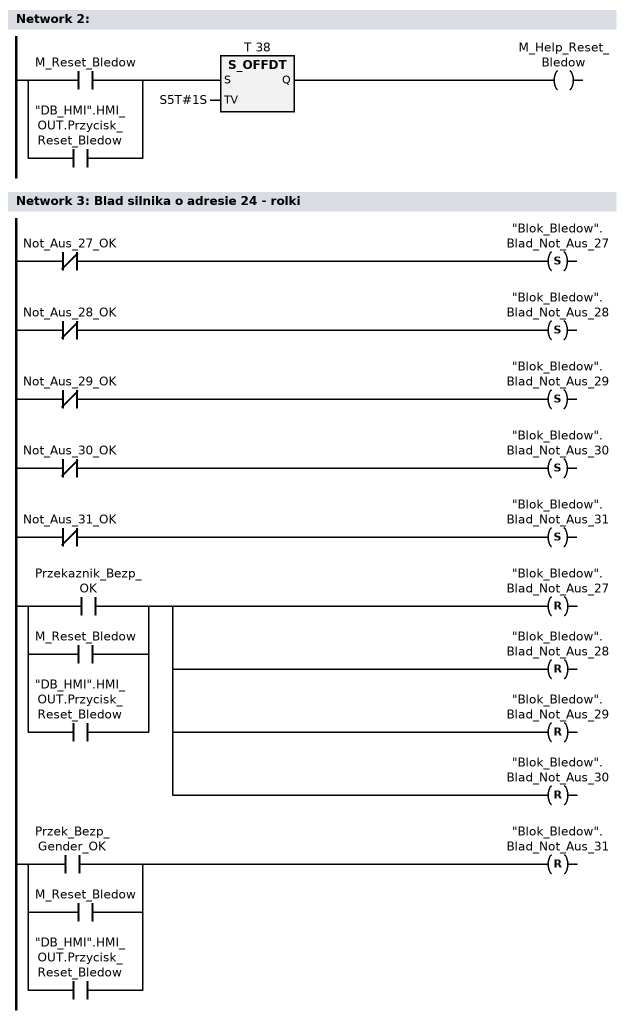
NETWORK
TITLE =
      A(;
      O     "M_Reset_Bledow";
      O     "DB_HMI".HMI_OUT.Przycisk_Reset_Bledow;
      );
      L     S5T#1S;
      SF    T 38;
      NOP   0;
      NOP   0;
      NOP   0;
      A     T 38;
      =     "M_Help_Reset_Bledow";
NETWORK
TITLE = Blad silnika o adresie 24 - rolki
//Bledy do panelu HMI
//Not Aus 27*******************************
      AN    "Not_Aus_27_OK";
      S     "Blok_Bledow".Blad_Not_Aus_27;
//Not Aus 28*******************************
      AN    "Not_Aus_28_OK";
      S     "Blok_Bledow".Blad_Not_Aus_28;
//Not Aus 29*******************************
      AN    "Not_Aus_29_OK";
      S     "Blok_Bledow".Blad_Not_Aus_29;
//Not Aus 30*******************************
      AN    "Not_Aus_30_OK";
      S     "Blok_Bledow".Blad_Not_Aus_30;
//Not Aus 31*******************************
      AN    "Not_Aus_31_OK";
      S     "Blok_Bledow".Blad_Not_Aus_31;
//Reset bledow not-aus
      O     "Przekaznik_Bezp_OK";
      O     "M_Reset_Bledow";
      O     "DB_HMI".HMI_OUT.Przycisk_Reset_Bledow;
      R     "Blok_Bledow".Blad_Not_Aus_27;
      R     "Blok_Bledow".Blad_Not_Aus_28;
      R     "Blok_Bledow".Blad_Not_Aus_29;
      R     "Blok_Bledow".Blad_Not_Aus_30;
      O     "Przek_Bezp_Gender_OK";
      O     "M_Reset_Bledow";
      O     "DB_HMI".HMI_OUT.Przycisk_Reset_Bledow;
      R     "Blok_Bledow".Blad_Not_Aus_31;
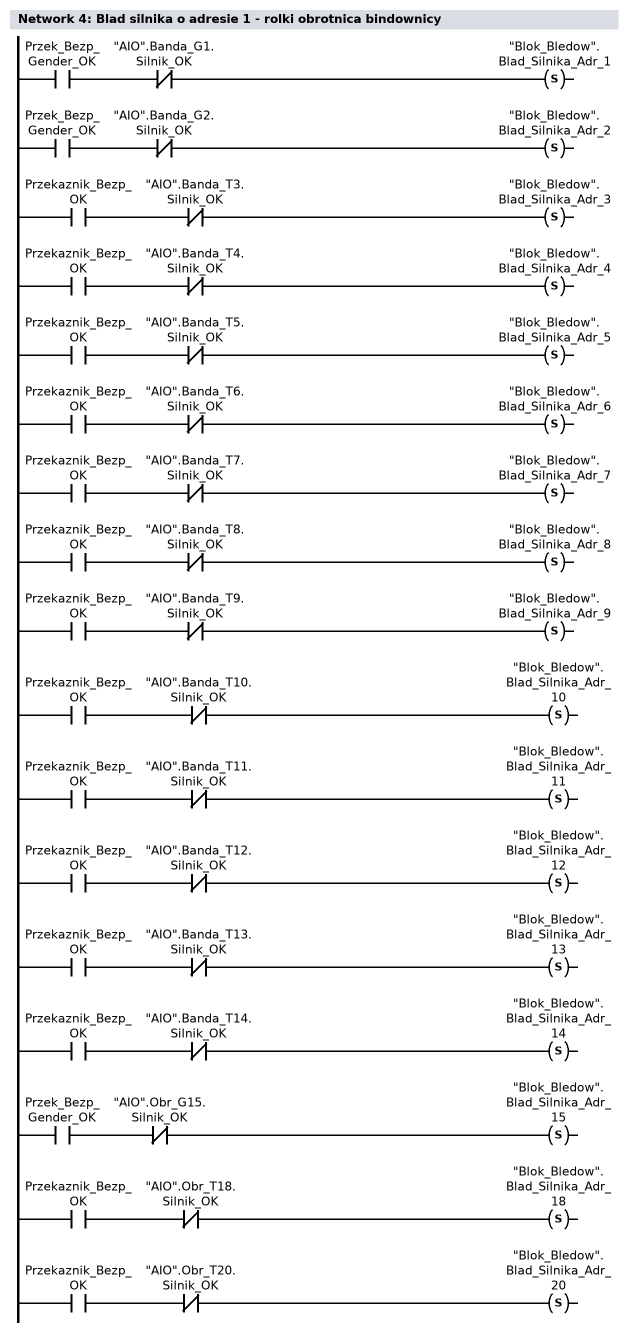
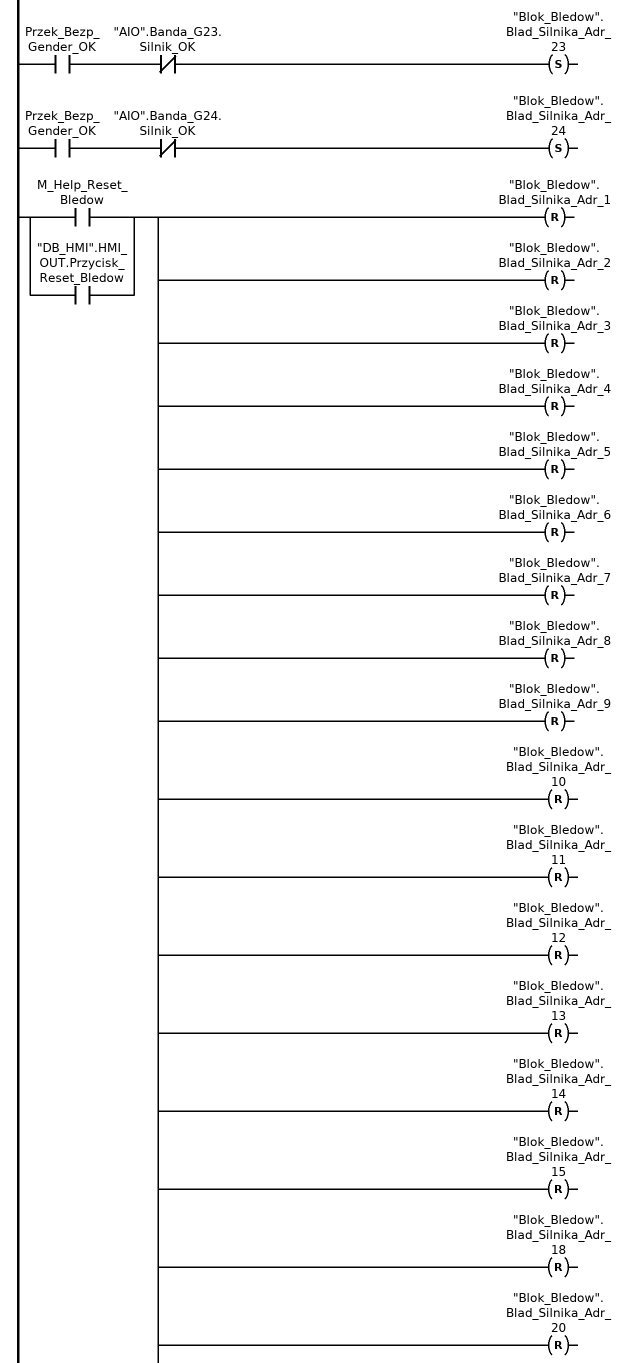
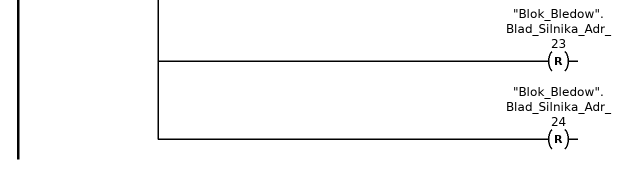
NETWORK
TITLE = Blad silnika o adresie 1 - rolki obrotnica bindownicy
//Bledy napedow
//Bledy napedow
      A     "Przek_Bezp_Gender_OK";
      AN    "AIO".Banda_G1.Silnik_OK;
      S     "Blok_Bledow".Blad_Silnika_Adr_1;
      A     "Przek_Bezp_Gender_OK";
      AN    "AIO".Banda_G2.Silnik_OK;
      S     "Blok_Bledow".Blad_Silnika_Adr_2;
      A     "Przekaznik_Bezp_OK";
      AN    "AIO".Banda_T3.Silnik_OK;
      S     "Blok_Bledow".Blad_Silnika_Adr_3;
      A     "Przekaznik_Bezp_OK";
      AN    "AIO".Banda_T4.Silnik_OK;
      S     "Blok_Bledow".Blad_Silnika_Adr_4;
      A     "Przekaznik_Bezp_OK";
      AN    "AIO".Banda_T5.Silnik_OK;
      S     "Blok_Bledow".Blad_Silnika_Adr_5;
      A     "Przekaznik_Bezp_OK";
      AN    "AIO".Banda_T6.Silnik_OK;
      S     "Blok_Bledow".Blad_Silnika_Adr_6;
      A     "Przekaznik_Bezp_OK";
      AN    "AIO".Banda_T7.Silnik_OK;
      S     "Blok_Bledow".Blad_Silnika_Adr_7;
      A     "Przekaznik_Bezp_OK";
      AN    "AIO".Banda_T8.Silnik_OK;
      S     "Blok_Bledow".Blad_Silnika_Adr_8;
      A     "Przekaznik_Bezp_OK";
      AN    "AIO".Banda_T9.Silnik_OK;
      S     "Blok_Bledow".Blad_Silnika_Adr_9;
      A     "Przekaznik_Bezp_OK";
      AN    "AIO".Banda_T10.Silnik_OK;
      S     "Blok_Bledow".Blad_Silnika_Adr_10;
      A     "Przekaznik_Bezp_OK";
      AN    "AIO".Banda_T11.Silnik_OK;
      S     "Blok_Bledow".Blad_Silnika_Adr_11;
      A     "Przekaznik_Bezp_OK";
      AN    "AIO".Banda_T12.Silnik_OK;
      S     "Blok_Bledow".Blad_Silnika_Adr_12;
      A     "Przekaznik_Bezp_OK";
      AN    "AIO".Banda_T13.Silnik_OK;
      S     "Blok_Bledow".Blad_Silnika_Adr_13;
      A     "Przekaznik_Bezp_OK";
      AN    "AIO".Banda_T14.Silnik_OK;
      S     "Blok_Bledow".Blad_Silnika_Adr_14;
      A     "Przek_Bezp_Gender_OK";
      AN    "AIO".Obr_G15.Silnik_OK;
      S     "Blok_Bledow".Blad_Silnika_Adr_15;
      A     "Przekaznik_Bezp_OK";
      AN    "AIO".Obr_T18.Silnik_OK;
      S     "Blok_Bledow".Blad_Silnika_Adr_18;
      A     "Przekaznik_Bezp_OK";
      AN    "AIO".Obr_T20.Silnik_OK;
      S     "Blok_Bledow".Blad_Silnika_Adr_20;
      A     "Przek_Bezp_Gender_OK";
      AN    "AIO".Banda_G23.Silnik_OK;
      S     "Blok_Bledow".Blad_Silnika_Adr_23;
      A     "Przek_Bezp_Gender_OK";
      AN    "AIO".Banda_G24.Silnik_OK;
      S     "Blok_Bledow".Blad_Silnika_Adr_24;
//Reset bledow napedow
//Reset bledow not-aus
      O     "M_Help_Reset_Bledow";
      O     "DB_HMI".HMI_OUT.Przycisk_Reset_Bledow;
      R     "Blok_Bledow".Blad_Silnika_Adr_1;
      R     "Blok_Bledow".Blad_Silnika_Adr_2;
      R     "Blok_Bledow".Blad_Silnika_Adr_3;
      R     "Blok_Bledow".Blad_Silnika_Adr_4;
      R     "Blok_Bledow".Blad_Silnika_Adr_5;
      R     "Blok_Bledow".Blad_Silnika_Adr_6;
      R     "Blok_Bledow".Blad_Silnika_Adr_7;
      R     "Blok_Bledow".Blad_Silnika_Adr_8;
      R     "Blok_Bledow".Blad_Silnika_Adr_9;
      R     "Blok_Bledow".Blad_Silnika_Adr_10;
      R     "Blok_Bledow".Blad_Silnika_Adr_11;
      R     "Blok_Bledow".Blad_Silnika_Adr_12;
      R     "Blok_Bledow".Blad_Silnika_Adr_13;
      R     "Blok_Bledow".Blad_Silnika_Adr_14;
      R     "Blok_Bledow".Blad_Silnika_Adr_15;
      R     "Blok_Bledow".Blad_Silnika_Adr_18;
      R     "Blok_Bledow".Blad_Silnika_Adr_20;
      R     "Blok_Bledow".Blad_Silnika_Adr_23;
      R     "Blok_Bledow".Blad_Silnika_Adr_24;
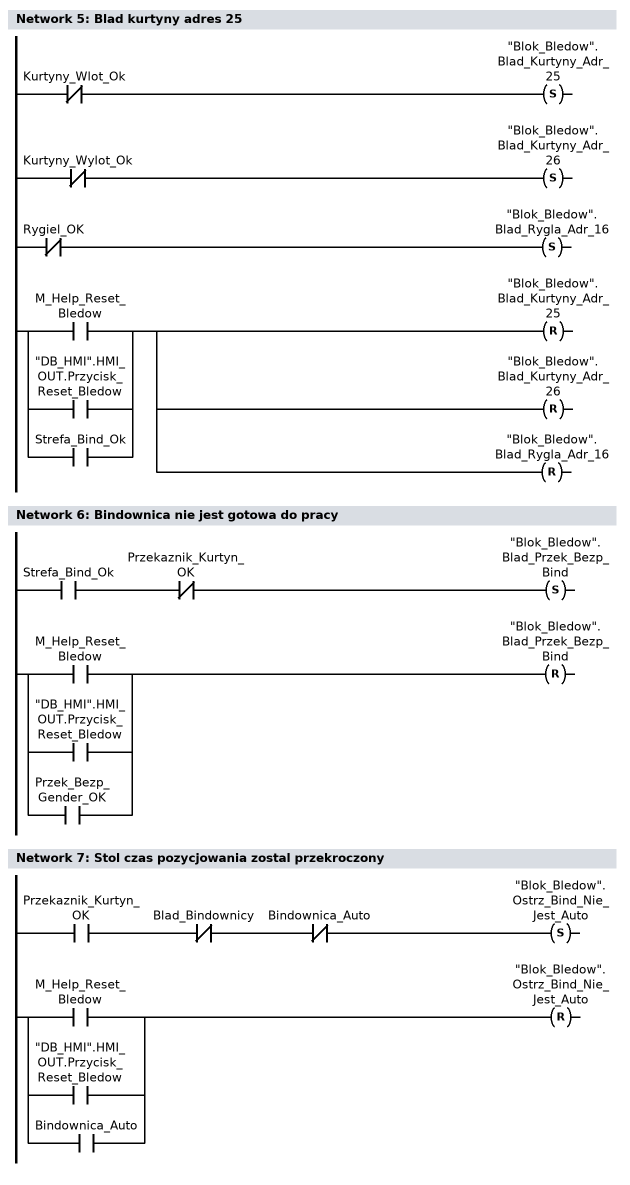
NETWORK
TITLE = Blad kurtyny adres 25
//Bledy kurtyn kasownie samoistne
      AN    "Kurtyny_Wlot_Ok";
      S     "Blok_Bledow".Blad_Kurtyny_Adr_25;
      AN    "Kurtyny_Wylot_Ok";
      S     "Blok_Bledow".Blad_Kurtyny_Adr_26;
      AN    "Rygiel_OK";
      S     "Blok_Bledow".Blad_Rygla_Adr_16;
      O     "M_Help_Reset_Bledow";
      O     "DB_HMI".HMI_OUT.Przycisk_Reset_Bledow;
      O     "Strefa_Bind_Ok";
      R     "Blok_Bledow".Blad_Kurtyny_Adr_25;
      R     "Blok_Bledow".Blad_Kurtyny_Adr_26;
      R     "Blok_Bledow".Blad_Rygla_Adr_16;
NETWORK
TITLE = Bindownica nie jest gotowa do pracy
//Blad Przekaznika bezpieczenstwa kurtyn
      A     "Strefa_Bind_Ok";
      AN    "Przekaznik_Kurtyn_OK";
      S     "Blok_Bledow".Blad_Przek_Bezp_Bind;
      O     "M_Help_Reset_Bledow";
      O     "DB_HMI".HMI_OUT.Przycisk_Reset_Bledow;
      O     "Przek_Bezp_Gender_OK";
      R     "Blok_Bledow".Blad_Przek_Bezp_Bind;
NETWORK
TITLE = Stol czas pozycjowania zostal przekroczony
//Blad informacyjny bindownica nie jest w auto
      A     "Przekaznik_Kurtyn_OK";
      AN    "Blad_Bindownicy";
      AN    "Bindownica_Auto";
      S     "Blok_Bledow".Ostrz_Bind_Nie_Jest_Auto;
      O     "M_Help_Reset_Bledow";
      O     "DB_HMI".HMI_OUT.Przycisk_Reset_Bledow;
      O     "Bindownica_Auto";
      R     "Blok_Bledow".Ostrz_Bind_Nie_Jest_Auto;
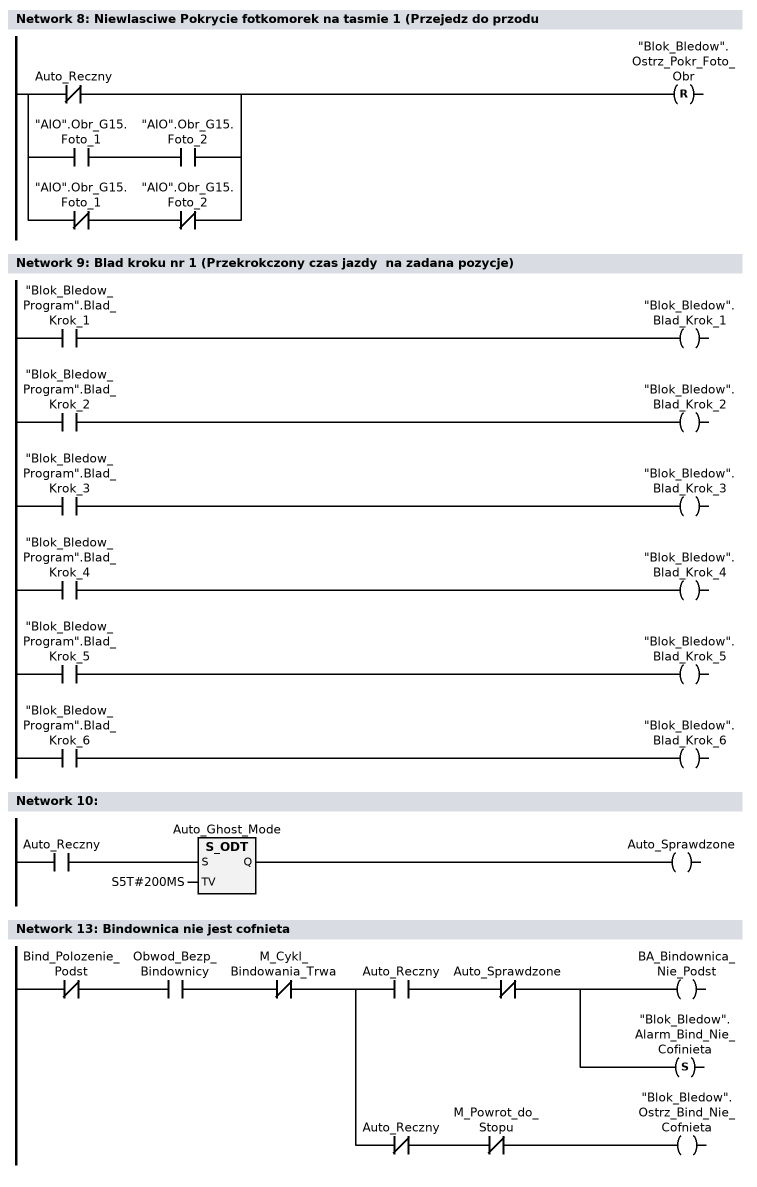
NETWORK
TITLE = Niewlasciwe Pokrycie fotkomorek na tasmie 1 (Przejedz do przodu 
//Ostrzezenie palety nie sa na fotokomorkach przednich
//
//Obrotnica
      ON    "Auto_Reczny";
      O;
      A     "AIO".Obr_G15.Foto_1;
      A     "AIO".Obr_G15.Foto_2;
      O;
      AN    "AIO".Obr_G15.Foto_1;
      AN    "AIO".Obr_G15.Foto_2;
      R     "Blok_Bledow".Ostrz_Pokr_Foto_Obr;
NETWORK
TITLE = Blad kroku nr 1 (Przekrokczony czas jazdy  na zadana pozycje)
//Bledy Zapalajaca czerwona lampke na panelu HMI
//Kwitowanie tych bledow przy pomocy przycisku. Reset nastepnie dalszy krok to 
//przywrocenie automatyki auto lub cyklem start
//
//
// Bledy czasu tranzycji krokow
      A     "Blok_Bledow_Program".Blad_Krok_1;
      =     "Blok_Bledow".Blad_Krok_1;
      A     "Blok_Bledow_Program".Blad_Krok_2;
      =     "Blok_Bledow".Blad_Krok_2;
      A     "Blok_Bledow_Program".Blad_Krok_3;
      =     "Blok_Bledow".Blad_Krok_3;
      A     "Blok_Bledow_Program".Blad_Krok_4;
      =     "Blok_Bledow".Blad_Krok_4;
      A     "Blok_Bledow_Program".Blad_Krok_5;
      =     "Blok_Bledow".Blad_Krok_5;
      A     "Blok_Bledow_Program".Blad_Krok_6;
      =     "Blok_Bledow".Blad_Krok_6;
NETWORK
TITLE =
//Wypadniecie maszyny z automatyki. Oraz powrot do polautomatu gdy automatyka nie 
//spelniona. 
      A     "Auto_Reczny";
      L     S5T#200MS;
      SD    "Auto_Ghost_Mode";
      NOP   0;
      NOP   0;
      NOP   0;
      A     "Auto_Ghost_Mode";
      =     "Auto_Sprawdzone";
NETWORK
TITLE =
NETWORK
TITLE =
//Warunki sprawdzane podczas 200ms trybu Ghost Mode
//bity m210 w gore
NETWORK
TITLE = Bindownica nie jest cofnieta
//Bindownica nie jest w pozycji podstawoej
      AN    "Bind_Polozenie_Podst";
      A     "Obwod_Bezp_Bindownicy";
      AN    "M_Cykl_Bindowania_Trwa";
      =     L 0.0;
      A     L 0.0;
      A     "Auto_Reczny";
      AN    "Auto_Sprawdzone";
      =     "BA_Bindownica_Nie_Podst";
      S     "Blok_Bledow".Alarm_Bind_Nie_Cofinieta;
      A     L 0.0;
      AN    "Auto_Reczny";
      AN    "M_Powrot_do_Stopu";
      =     "Blok_Bledow".Ostrz_Bind_Nie_Cofnieta;
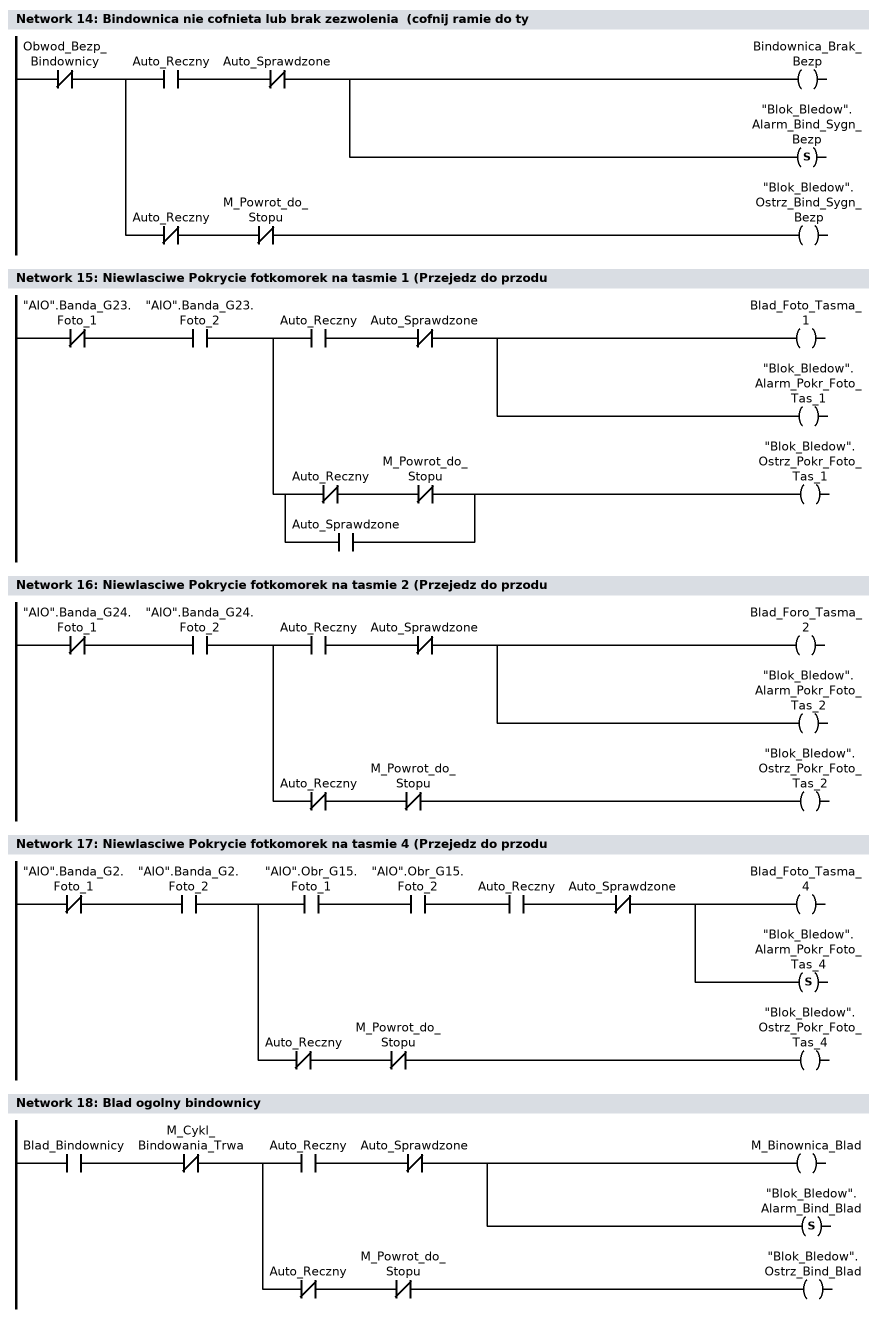
NETWORK
TITLE = Bindownica nie cofnieta lub brak zezwolenia  (cofnij ramie do ty
//Bindownica nie daje sygnalu bezpieczestwa
      AN    "Obwod_Bezp_Bindownicy";
      =     L 0.0;
      A     L 0.0;
      A     "Auto_Reczny";
      AN    "Auto_Sprawdzone";
      =     "Bindownica_Brak_Bezp";
      S     "Blok_Bledow".Alarm_Bind_Sygn_Bezp;
      A     L 0.0;
      AN    "Auto_Reczny";
      AN    "M_Powrot_do_Stopu";
      =     "Blok_Bledow".Ostrz_Bind_Sygn_Bezp;
NETWORK
TITLE = Niewlasciwe Pokrycie fotkomorek na tasmie 1 (Przejedz do przodu 
//Tasma 1 Wyjatek bo tutaj kladzie sie palete w automacie przez wozek
      AN    "AIO".Banda_G23.Foto_1;
      A     "AIO".Banda_G23.Foto_2;
      =     L 0.0;
      A     L 0.0;
      A     "Auto_Reczny";
      AN    "Auto_Sprawdzone";
      =     "Blad_Foto_Tasma_1";
      =     "Blok_Bledow".Alarm_Pokr_Foto_Tas_1;
      A     L 0.0;
      A(;
      AN    "Auto_Reczny";
      AN    "M_Powrot_do_Stopu";
      O     "Auto_Sprawdzone";
      );
      =     "Blok_Bledow".Ostrz_Pokr_Foto_Tas_1;
NETWORK
TITLE = Niewlasciwe Pokrycie fotkomorek na tasmie 2 (Przejedz do przodu 
//Tasma 2   O     "DB_HMI".HMI_OUT.Przycisk_Reset_Bledow
      AN    "AIO".Banda_G24.Foto_1;
      A     "AIO".Banda_G24.Foto_2;
      =     L 0.0;
      A     L 0.0;
      A     "Auto_Reczny";
      AN    "Auto_Sprawdzone";
      =     "Blad_Foro_Tasma_2";
      =     "Blok_Bledow".Alarm_Pokr_Foto_Tas_2;
      A     L 0.0;
      AN    "Auto_Reczny";
      AN    "M_Powrot_do_Stopu";
      =     "Blok_Bledow".Ostrz_Pokr_Foto_Tas_2;
NETWORK
TITLE = Niewlasciwe Pokrycie fotkomorek na tasmie 4 (Przejedz do przodu 
//Tasma:4      "DB_HMI".HMI_OUT.Przycisk_Reset_Bledow
      AN    "AIO".Banda_G2.Foto_1;
      A     "AIO".Banda_G2.Foto_2;
      =     L 0.0;
      A     L 0.0;
      A     "AIO".Obr_G15.Foto_1;
      A     "AIO".Obr_G15.Foto_2;
      A     "Auto_Reczny";
      AN    "Auto_Sprawdzone";
      =     "Blad_Foto_Tasma_4";
      S     "Blok_Bledow".Alarm_Pokr_Foto_Tas_4;
      A     L 0.0;
      AN    "Auto_Reczny";
      AN    "M_Powrot_do_Stopu";
      =     "Blok_Bledow".Ostrz_Pokr_Foto_Tas_4;
NETWORK
TITLE = Blad ogolny bindownicy 
//Blad ogolny bindownicy
      A     "Blad_Bindownicy";
      AN    "M_Cykl_Bindowania_Trwa";
      =     L 0.0;
      A     L 0.0;
      A     "Auto_Reczny";
      AN    "Auto_Sprawdzone";
      =     "M_Binownica_Blad";
      S     "Blok_Bledow".Alarm_Bind_Blad;
      A     L 0.0;
      AN    "Auto_Reczny";
      AN    "M_Powrot_do_Stopu";
      =     "Blok_Bledow".Ostrz_Bind_Blad;
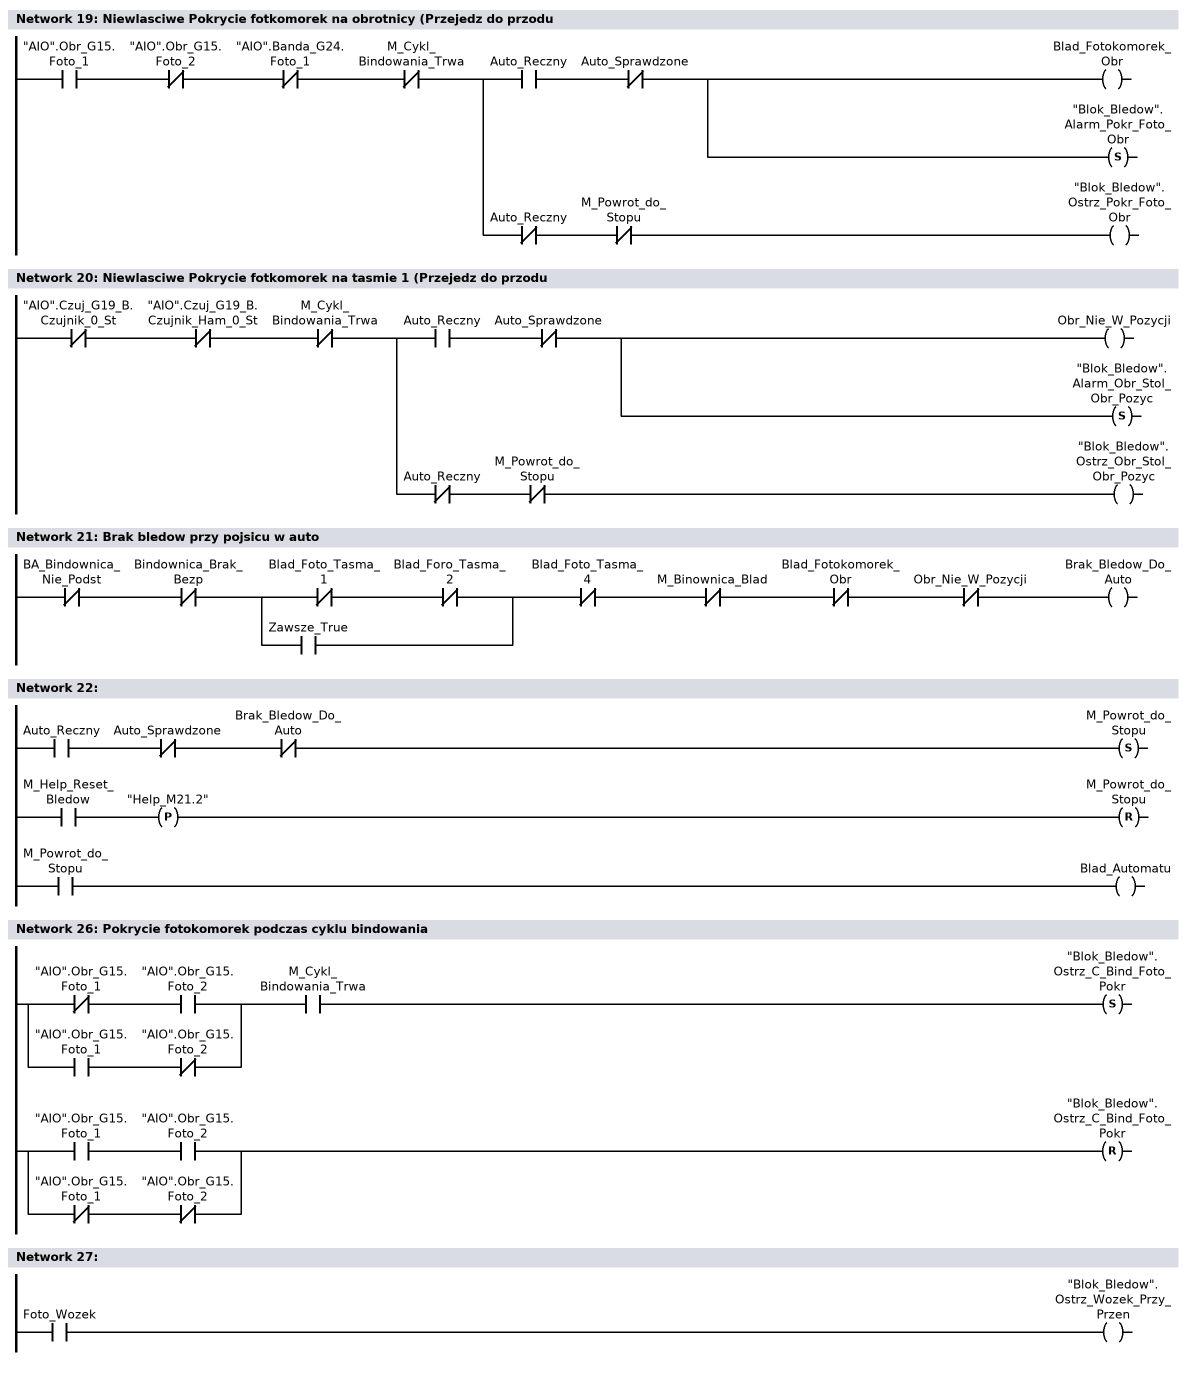
NETWORK
TITLE = Niewlasciwe Pokrycie fotkomorek na obrotnicy (Przejedz do przodu
//Blad fotokomorek stolu obrotowego
      A     "AIO".Obr_G15.Foto_1;
      AN    "AIO".Obr_G15.Foto_2;
      AN    "AIO".Banda_G24.Foto_1;
      AN    "M_Cykl_Bindowania_Trwa";
      =     L 0.0;
      A     L 0.0;
      A     "Auto_Reczny";
      AN    "Auto_Sprawdzone";
      =     "Blad_Fotokomorek_Obr";
      S     "Blok_Bledow".Alarm_Pokr_Foto_Obr;
      A     L 0.0;
      AN    "Auto_Reczny";
      AN    "M_Powrot_do_Stopu";
      =     "Blok_Bledow".Ostrz_Pokr_Foto_Obr;
NETWORK
TITLE = Niewlasciwe Pokrycie fotkomorek na tasmie 1 (Przejedz do przodu 
//Stol obrotowy nie w pozycji
      AN    "AIO".Czuj_G19_B.Czujnik_0_St;
      AN    "AIO".Czuj_G19_B.Czujnik_Ham_0_St;
      AN    "M_Cykl_Bindowania_Trwa";
      =     L 0.0;
      A     L 0.0;
      A     "Auto_Reczny";
      AN    "Auto_Sprawdzone";
      =     "Obr_Nie_W_Pozycji";
      S     "Blok_Bledow".Alarm_Obr_Stol_Obr_Pozyc;
      A     L 0.0;
      AN    "Auto_Reczny";
      AN    "M_Powrot_do_Stopu";
      =     "Blok_Bledow".Ostrz_Obr_Stol_Obr_Pozyc;
NETWORK
TITLE = Brak bledow przy pojsicu w auto
//Sprawdzam
      AN    "BA_Bindownica_Nie_Podst";
      AN    "Bindownica_Brak_Bezp";
      A(;
      AN    "Blad_Foto_Tasma_1";
      AN    "Blad_Foro_Tasma_2";
      O     "Zawsze_True";
      );
      AN    "Blad_Foto_Tasma_4";
      AN    "M_Binownica_Blad";
      AN    "Blad_Fotokomorek_Obr";
      AN    "Obr_Nie_W_Pozycji";
      =     "Brak_Bledow_Do_Auto";
NETWORK
TITLE =
//Powrot do stopu polautomatu jesli jest blad
      A     "Auto_Reczny";
      AN    "Auto_Sprawdzone";
      AN    "Brak_Bledow_Do_Auto";
      S     "M_Powrot_do_Stopu";
      A     "M_Help_Reset_Bledow";
      FP    "Help_M21.2";
      R     "M_Powrot_do_Stopu";
      A     "M_Powrot_do_Stopu";
      =     "Blad_Automatu";
NETWORK
TITLE = Bindownica nie cofnieta lub brak zezwolenia  (cofnij ramie do ty
//reset komunikatow
//
      A     "M_Help_Reset_Bledow";
//Alarmy
      R     "Blok_Bledow".Alarm_Obr_Stol_Obr_Pozyc;
      R     "Blok_Bledow".Alarm_Bind_Nie_Cofinieta;
      R     "Blok_Bledow".Alarm_Bind_Sygn_Bezp;
      R     "Blok_Bledow".rez3;
      R     "Blok_Bledow".rez_6_0;
      R     "Blok_Bledow".Alarm_Pokr_Foto_Tas_1;
      R     "Blok_Bledow".Alarm_Pokr_Foto_Tas_2;
      R     "Blok_Bledow".Alarm_Pokr_Foto_Tas_4;
      R     "Blok_Bledow".Alarm_Pokr_Foto_Obr;
      R     "Blok_Bledow".Alarm_Bind_Nie_Jest_Auto;
      R     "Blok_Bledow".Alarm_Bind_Blad;
      R     "Blok_Bledow".rez_6_7;
      R     "Blok_Bledow".Ostrz_Prasa_Nie_W_Gorze;
      R     "Blok_Bledow".rez_7_1;
//Warnings
      R     "Blok_Bledow".Ostrz_Bind_Blad;
      R     "Blok_Bledow".Ostrz_Bind_Nie_Cofnieta;
      R     "Blok_Bledow".Ostrz_Bind_Sygn_Bezp;
      R     "Blok_Bledow".Ostrz_Bind_Nie_Jest_Auto;
      R     "Blok_Bledow".Ostrz_Stol_Obr_Foto;
      R     "Blok_Bledow".Ostrz_Obr_Stol_Obr_Pozyc;
      R     "Blok_Bledow".Ostrz_Pokr_Foto_Tas_1;
      R     "Blok_Bledow".Ostrz_Pokr_Foto_Tas_2;
      R     "Blok_Bledow".Ostrz_Pokr_Foto_Obr;
      R     "Blok_Bledow".Ostrz_Pokr_Foto_Tas_4;
      CLR;
NETWORK
TITLE =
//Koniec sprawdzanie wejscia w automatyke
NETWORK
TITLE =
//Sprawdzenie maszyny podczas cyklu. Zwracane sa ostrzezenia by byla informacja 
//ale nie przerwac dzialania
NETWORK
TITLE = Pokrycie fotokomorek podczas cyklu bindowania
//Niewlasciwe pokrycie fotokomorek podczas cyklu
      A(;
      AN    "AIO".Obr_G15.Foto_1;
      A     "AIO".Obr_G15.Foto_2;
      O;
      A     "AIO".Obr_G15.Foto_1;
      AN    "AIO".Obr_G15.Foto_2;
      );
      A     "M_Cykl_Bindowania_Trwa";
      S     "Blok_Bledow".Ostrz_C_Bind_Foto_Pokr;
      A(;
      A     "AIO".Obr_G15.Foto_1;
      A     "AIO".Obr_G15.Foto_2;
      O;
      AN    "AIO".Obr_G15.Foto_1;
      AN    "AIO".Obr_G15.Foto_2;
      );
      R     "Blok_Bledow".Ostrz_C_Bind_Foto_Pokr;
      NOP   0;
NETWORK
TITLE =
//Cykl trwa a bindownica nie jest z tylu
      A     "Foto_Wozek";
      =     "Blok_Bledow".Ostrz_Wozek_Przy_Przen;
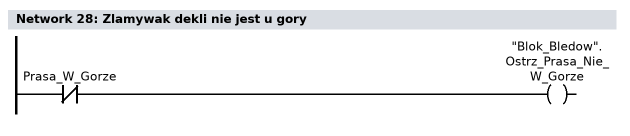
NETWORK
TITLE = Zlamywak dekli nie jest u gory 
      AN    "Prasa_W_Gorze";
      =     "Blok_Bledow".Ostrz_Prasa_Nie_W_Gorze;
END_FUNCTION

FUNCTION "FC_HMI" : VOID	// FC 120
VERSION : 0.1
VAR_TEMP
  LW0_Help : INT ;
END_VAR
BEGIN
NETWORK
TITLE =
//Ten network celowo wolny
NETWORK
TITLE = Tryb Pracy Wiazanie poprzeczne
//Wybranie trybu pracy resetuje pozostale tryby pracy
//1-Przelot
//Offline************************************
      A     "DB_HMI".HMI_IN_OUT.Tp_Przelot;
      AN    "Linia_Gender_ONline";
      R     "DB_HMI".HMI_IN_OUT.Tp_Wiazanie_Poprzeczne;
      R     "DB_HMI".HMI_IN_OUT.Tp_Wiazanie_Wzdluzne;
      R     "DB_HMI".HMI_IN_OUT.Tp_Wiazanie_Pop_Wzdl;
//*
      R     "Blok_Para".Wiazanie_Poprzeczne;
      R     "Blok_Para".Wiazanie_Wzdluzne;
//Online*************************************
      AN    "ON_Wiazanie_Poprzeczne";
      AN    "ON_Wiazanie_Wzdluzne";
      A     "Linia_Gender_ONline";
      R     "DB_HMI".HMI_IN_OUT.Tp_Wiazanie_Poprzeczne;
      R     "DB_HMI".HMI_IN_OUT.Tp_Wiazanie_Wzdluzne;
      R     "DB_HMI".HMI_IN_OUT.Tp_Wiazanie_Pop_Wzdl;
//*
      R     "Blok_Para".Wiazanie_Poprzeczne;
      R     "Blok_Para".Wiazanie_Wzdluzne;
NETWORK
TITLE = Tryb Pracy Wiazanie poprzeczne
//Wybranie trybu pracy resetuje pozostale tryby pracy
//2-Wiazanie Poprzeczne
//Offline************************************
      A     "DB_HMI".HMI_IN_OUT.Tp_Wiazanie_Poprzeczne;
      AN    "Linia_Gender_ONline";
      R     "DB_HMI".HMI_IN_OUT.Tp_Przelot;
      R     "DB_HMI".HMI_IN_OUT.Tp_Wiazanie_Wzdluzne;
      R     "DB_HMI".HMI_IN_OUT.Tp_Wiazanie_Pop_Wzdl;
//*
      S     "Blok_Para".Wiazanie_Poprzeczne;
      R     "Blok_Para".Wiazanie_Wzdluzne;
//Online*************************************
      A     "ON_Wiazanie_Poprzeczne";
      AN    "ON_Wiazanie_Wzdluzne";
      A     "Linia_Gender_ONline";
      R     "DB_HMI".HMI_IN_OUT.Tp_Przelot;
      R     "DB_HMI".HMI_IN_OUT.Tp_Wiazanie_Wzdluzne;
      R     "DB_HMI".HMI_IN_OUT.Tp_Wiazanie_Pop_Wzdl;
//*
      S     "Blok_Para".Wiazanie_Poprzeczne;
      R     "Blok_Para".Wiazanie_Wzdluzne;
NETWORK
TITLE = Tryb Pracy Wiazanie poprzeczne
//Wybranie trybu pracy resetuje pozostale tryby pracy
//3-Wiazanie Wzdluzne
//Offline************************************
      A     "DB_HMI".HMI_IN_OUT.Tp_Wiazanie_Wzdluzne;
      AN    "Linia_Gender_ONline";
      R     "DB_HMI".HMI_IN_OUT.Tp_Przelot;
      R     "DB_HMI".HMI_IN_OUT.Tp_Wiazanie_Poprzeczne;
      R     "DB_HMI".HMI_IN_OUT.Tp_Wiazanie_Pop_Wzdl;
//*
      R     "Blok_Para".Wiazanie_Poprzeczne;
      S     "Blok_Para".Wiazanie_Wzdluzne;
//Online*************************************
      AN    "ON_Wiazanie_Poprzeczne";
      A     "ON_Wiazanie_Wzdluzne";
      A     "Linia_Gender_ONline";
      R     "DB_HMI".HMI_IN_OUT.Tp_Przelot;
      R     "DB_HMI".HMI_IN_OUT.Tp_Wiazanie_Poprzeczne;
      R     "DB_HMI".HMI_IN_OUT.Tp_Wiazanie_Pop_Wzdl;
//*
      R     "Blok_Para".Wiazanie_Poprzeczne;
      S     "Blok_Para".Wiazanie_Wzdluzne;
NETWORK
TITLE = Tryb Pracy Wiazanie poprzeczne
//Wybranie trybu pracy resetuje pozostale tryby pracy
//4-Wiazanie Poprzeczne i wzdluzne
//Offline************************************
      A     "DB_HMI".HMI_IN_OUT.Tp_Wiazanie_Pop_Wzdl;
      AN    "Linia_Gender_ONline";
      R     "DB_HMI".HMI_IN_OUT.Tp_Przelot;
      R     "DB_HMI".HMI_IN_OUT.Tp_Wiazanie_Poprzeczne;
      R     "DB_HMI".HMI_IN_OUT.Tp_Wiazanie_Wzdluzne;
//*
      S     "Blok_Para".Wiazanie_Poprzeczne;
      S     "Blok_Para".Wiazanie_Wzdluzne;
//Online*************************************
      A     "ON_Wiazanie_Poprzeczne";
      A     "ON_Wiazanie_Wzdluzne";
      A     "Linia_Gender_ONline";
      R     "DB_HMI".HMI_IN_OUT.Tp_Przelot;
      R     "DB_HMI".HMI_IN_OUT.Tp_Wiazanie_Poprzeczne;
      R     "DB_HMI".HMI_IN_OUT.Tp_Wiazanie_Wzdluzne;
//*
      S     "Blok_Para".Wiazanie_Poprzeczne;
      S     "Blok_Para".Wiazanie_Wzdluzne;
NETWORK
TITLE = wybrano tryb pracy przelot
      AN    "Blok_Para".Wiazanie_Wzdluzne;
      AN    "Blok_Para".Wiazanie_Poprzeczne;
      =     "DB_HMI".HMI_IN.Wybrano_TP_Przelot;
//-wzdl
      A     "Blok_Para".Wiazanie_Wzdluzne;
      AN    "Blok_Para".Wiazanie_Poprzeczne;
      =     "DB_HMI".HMI_IN.Wybrano_TP_Wiazanie_Wzdl;
//-pop
      AN    "Blok_Para".Wiazanie_Wzdluzne;
      A     "Blok_Para".Wiazanie_Poprzeczne;
      =     "DB_HMI".HMI_IN.Wybrano_TP_Wiazanie_Pop;
//-pop -wzdl
      A     "Blok_Para".Wiazanie_Wzdluzne;
      A     "Blok_Para".Wiazanie_Poprzeczne;
      =     "DB_HMI".HMI_IN.Wybrano_TP_Wiazanie_Krzy;
NETWORK
TITLE =
//znacznik trybu wiazania
//krok_1  - przelot
      A     "DB_HMI".HMI_IN.Wybrano_TP_Przelot;
      L     1;
      JC    ztw;
//krok_2 - wzdluzna
      A     "DB_HMI".HMI_IN.Wybrano_TP_Wiazanie_Wzdl;
      L     2;
      JC    ztw;
//krok_3 - poprzeczne
      A     "DB_HMI".HMI_IN.Wybrano_TP_Wiazanie_Pop;
      L     3;
      JC    ztw;
//krok_4 - krzyzowe
      A     "DB_HMI".HMI_IN.Wybrano_TP_Wiazanie_Krzy;
      L     4;
      JC    ztw;
//daj 0
ztw:  T     "DB_HMI".HMI_IN.tryb_wiaz;
NETWORK
TITLE = Tryb Pracy Wiazanie wzduzne
//Zalaczenie Pozycjonowania
      A     "DB_HMI".HMI_IN_OUT.Tp_Pozycjonowanie;
      S     "Blok_Para".Pozycjonowanie;
      AN    "DB_HMI".HMI_IN_OUT.Tp_Pozycjonowanie;
      R     "Blok_Para".Pozycjonowanie;
      NOP   0;
NETWORK
TITLE = fotokomorka hamowania obrotnicy do kata 0st
//Fotokomorki katow pozycjonowania obrotnicy
      A     "AIO".Czuj_G19_B.Czujnik_Ham_0_St;
      =     "DB_HMI".HMI_IN.Czujnik_Ham_0_St;
      A     "AIO".Czuj_G19_B.Czujnik_0_St;
      =     "DB_HMI".HMI_IN.Czujnik_0_St;
      A     "AIO".Czuj_G19_B.Czujnik_Ham_90_St;
      =     "DB_HMI".HMI_IN.Czujnik_Ham_90_St;
      A     "AIO".Czuj_G19_B.Czujnik_90_St;
      =     "DB_HMI".HMI_IN.Czujnik_90_St;
      A     "AIO".Czuj_G17_B.Czujnik_Ham_180_St;
      =     "DB_HMI".HMI_IN.Czujnik_Ham_180_St;
      A     "AIO".Czuj_G17_B.Czujnik_180_St;
      =     "DB_HMI".HMI_IN.Czujnik_180_St;
      A     "AIO".Czuj_G17_B.Czujnik_Ham_270_St;
      =     "DB_HMI".HMI_IN.Czujnik_Ham_270_St;
      A     "AIO".Czuj_G17_B.Czujnik_270_St;
      =     "DB_HMI".HMI_IN.Czujnik_270_St;
NETWORK
TITLE = foto przednie bandzie wlotowej
//Fotokommorki
      A     "AIO".Banda_G23.Foto_1;
      =     "DB_HMI".HMI_IN.Foto_Tasma_1_Przod;
      A     "AIO".Banda_G23.Foto_2;
      =     "DB_HMI".HMI_IN.Foto_Tasma_1_Tyl;
      A     "AIO".Banda_G24.Foto_1;
      =     "DB_HMI".HMI_IN.Foto_Tasma_2_Przod;
      A     "AIO".Banda_G24.Foto_2;
      =     "DB_HMI".HMI_IN.Foto_Tasma_2_Tyl;
      A     "AIO".Obr_G15.Foto_1;
      =     "DB_HMI".HMI_IN.Foto_Obrotnica_3_Przod;
      A     "AIO".Obr_G15.Foto_2;
      =     "DB_HMI".HMI_IN.Foto_Obrotnica_3_Tyl;
      A     "AIO".Banda_G2.Foto_1;
      =     "DB_HMI".HMI_IN.Foto_Tasma_4_Przod;
      A     "AIO".Banda_G2.Foto_2;
      =     "DB_HMI".HMI_IN.Foto_Tasma_4_Tyl;
NETWORK
TITLE = tasma 1
//do wizualizacji przemieszczania palety na tasmie 1
      AN    "AIO".Banda_G23.Foto_1;
      A     "AIO".Banda_G23.Foto_2;
      =     "DB_HMI".HMI_IN.Paleta_na_Tasmie_1_T;
      A     "AIO".Banda_G23.Foto_1;
      AN    "AIO".Banda_G23.Foto_2;
      AN    "AIO".Banda_G24.Foto_2;
      =     "DB_HMI".HMI_IN.Paleta_na_Tasmie_1_P;
      A     "AIO".Banda_G23.Foto_1;
      A     "AIO".Banda_G23.Foto_2;
      =     "DB_HMI".HMI_IN.Paleta_na_Tasmie_1;
NETWORK
TITLE = tasma 2
//do wizualizacji przemieszczania palety na tasmie 2
      AN    "AIO".Banda_G24.Foto_1;
      A     "AIO".Banda_G24.Foto_2;
      =     "DB_HMI".HMI_IN.Paleta_na_Tasmie_2_T;
      A     "AIO".Banda_G24.Foto_1;
      AN    "AIO".Banda_G24.Foto_2;
      AN    "AIO".Obr_G15.Foto_1;
      =     "DB_HMI".HMI_IN.Paleta_na_Tasmie_2_P;
      A     "AIO".Banda_G24.Foto_1;
      A     "AIO".Banda_G24.Foto_2;
      =     "DB_HMI".HMI_IN.Paleta_na_Tasmie_2;
NETWORK
TITLE = tasma 3 (obrotnica)
//do wizualizacji przemieszczania palety na tasmie 3
      A     "AIO".Obr_G15.Foto_1;
      AN    "AIO".Obr_G15.Foto_2;
      A     "DB_HMI".HMI_IN.Czujnik_0_St;
      =     "DB_HMI".HMI_IN.Paleta_na_Tasmie_3_T;
      AN    "AIO".Obr_G15.Foto_1;
      A     "AIO".Obr_G15.Foto_2;
      AN    "AIO".Banda_G2.Foto_2;
      A     "DB_HMI".HMI_IN.Czujnik_0_St;
      =     "DB_HMI".HMI_IN.Paleta_na_Tasmie_3_P;
      A     "AIO".Obr_G15.Foto_1;
      A     "AIO".Obr_G15.Foto_2;
      A(;
      O     "DB_HMI".HMI_IN.Czujnik_0_St;
      O     "DB_HMI".HMI_IN.Czujnik_180_St;
      );
      =     "DB_HMI".HMI_IN.Paleta_na_Tasmie_3_0_180;
      A     "AIO".Obr_G15.Foto_1;
      A     "AIO".Obr_G15.Foto_2;
      A(;
      O     "DB_HMI".HMI_IN.Czujnik_90_St;
      O     "DB_HMI".HMI_IN.Czujnik_270_St;
      );
      =     "DB_HMI".HMI_IN.Paleta_na_Tasmie_3_90_27;
NETWORK
TITLE = tasma 4
//do wizualizacji przemieszczania palety na tasmie 4
      AN    "AIO".Banda_G2.Foto_1;
      A     "AIO".Banda_G2.Foto_2;
      =     "DB_HMI".HMI_IN.Paleta_na_Tasmie_4_T;
      A     "AIO".Banda_G2.Foto_1;
      AN    "AIO".Banda_G2.Foto_2;
      =     "DB_HMI".HMI_IN.Paleta_na_Tasmie_4_P;
      A     "AIO".Banda_G2.Foto_1;
      A     "AIO".Banda_G2.Foto_2;
      =     "DB_HMI".HMI_IN.Paleta_na_Tasmie_4;
NETWORK
TITLE = motor obrotnica 3 counter clock wise
//Napedy band
      A     "AIO".Obr_G15.CC_Wise;
      =     "DB_HMI".HMI_IN.Motor_Obrotnica_3_CCW;
      A     "AIO".Obr_G15.C_Wise;
      =     "DB_HMI".HMI_IN.Motor_Obrotnica_3_CW;
      A     "AIO".Banda_G23.CC_Wise;
      =     "DB_HMI".HMI_IN.Motor_Tasma_1_Przod;
      A     "AIO".Banda_G23.C_Wise;
      =     "DB_HMI".HMI_IN.Motor_Tasma_1_Tyl;
      A     "AIO".Banda_G24.C_Wise;
      =     "DB_HMI".HMI_IN.Motor_Tasma_2_Przod;
      A     "AIO".Banda_G24.CC_Wise;
      =     "DB_HMI".HMI_IN.Motor_Tasma_2_Tyl;
      A     "AIO".Banda_G1.C_Wise;
      =     "DB_HMI".HMI_IN.Motor_Tasma_3_Przod;
      A     "AIO".Banda_G1.CC_Wise;
      =     "DB_HMI".HMI_IN.Motor_Tasma_3_Tyl;
      A     "AIO".Banda_G2.CC_Wise;
      =     "DB_HMI".HMI_IN.Motor_Tasma_4_Przod;
      A     "AIO".Banda_G2.C_Wise;
      =     "DB_HMI".HMI_IN.Motor_Tasma_4_Tyl;
NETWORK
TITLE = obwod bezpieczenstwa bindownicy
//sygnaly wymiany danych pomiedzy transportem palet a bindownica
      A     "Obwod_Bezp_Bindownicy";
      =     "DB_HMI".HMI_IN.Interfefs_B_do_TP_B1;
      A     "Bind_Polozenie_Podst";
      =     "DB_HMI".HMI_IN.Interfefs_B_do_TP_B2;
      A     "Start_Koniec_Wiazania";
      =     "DB_HMI".HMI_IN.Interfefs_B_do_TP_B3;
      A     "Bindownica_Auto";
      =     "DB_HMI".HMI_IN.Interfefs_B_do_TP_B4;
      A     "Blad_Bindownicy";
      =     "DB_HMI".HMI_IN.Interfefs_B_do_TP_B5;
//Transport do bindownicy 
      A     "Wirt_Syg_Bezp_Gender";
      =     "DB_HMI".HMI_IN.Interfefs_TP_do_B_TP1;
      A     "Zezw_na_prace_Bind";
      =     "DB_HMI".HMI_IN.Interfefs_TP_do_B_TP2;
      A     "o_Start_Wiazania";
      =     "DB_HMI".HMI_IN.Interfefs_TP_do_B_TP3;
NETWORK
TITLE = przycisk zalaczenie Strefy bezpieczenstwa
//przyciski, przelaczniki kierunkow i lampki na panelu
      A     "pb_Strefa_bezpieczenstwa";
      =     "DB_HMI".HMI_IN.PB_Strefa_bezpieczenstwa;
      A     "pb_Reczny";
      =     "DB_HMI".HMI_IN.PB_Reczny;
      A     "pb_Auto";
      =     "DB_HMI".HMI_IN.PB_Auto;
      A     "pb_Reset";
      =     "DB_HMI".HMI_IN.PB_Reset;
      A     "pb_Stop";
      =     "DB_HMI".HMI_IN.PB_Stop;
      A     "pb_Cykl_Start";
      =     "DB_HMI".HMI_IN.PB_Cykl_Start;
      A     "pb_Wozek_Tyl";
      =     "DB_HMI".HMI_IN.PB_Tasma1_Tyl;
      A     "pb_Wozek_Przod";
      =     "DB_HMI".HMI_IN.PB_Tasma1_Przod;
      A     "pb_Tasma_1_Tyl";
      =     "DB_HMI".HMI_IN.PB_Tasma2_Tyl;
      A     "pb_Tasma_1_Przod";
      =     "DB_HMI".HMI_IN.PB_Tasma2_Przod;
      A     "pb_Tasma_2_Tyl";
      =     "DB_HMI".HMI_IN.PB_Tasma3_Tyl;
      A     "pb_Tasma_2_Przod";
      =     "DB_HMI".HMI_IN.PB_Tasma3_Przod;
      A     "pb_Tasma_Obr_Tyl";
      =     "DB_HMI".HMI_IN.PB_Tasma4_Tyl;
      A     "pb_Tasma_Obr_Przod";
      =     "DB_HMI".HMI_IN.PB_Tasma4_Przod;
      A     "pb_Tasma_Wylot_Przod";
      =     "DB_HMI".HMI_IN.PB_Tasma3_Obr_CW;
      A     "pb_Tasma_Wylot_Tyl";
      =     "DB_HMI".HMI_IN.PB_Tasma3_Obr_CCW;
      A     "Lampka_Blad_Bind";
      =     "DB_HMI".HMI_IN.Lampka_Blad_Bind;
      A     "Lampka_Strzal";
      =     "DB_HMI".HMI_IN.Lampka_Strzal_Tasmy;
      A     "Lampka_pb_Strefa_Bezp";
      =     "DB_HMI".HMI_IN.Lampka_Strefa_Bezp;
      A     "Lampka_pb_Reczny";
      =     "DB_HMI".HMI_IN.Lampka_PB_Reczny;
      A     "Lampka_pb_Auto";
      =     "DB_HMI".HMI_IN.Lampka_PB_Auto;
      A     "Lampka_pb_Reset";
      =     "DB_HMI".HMI_IN.Lampka_PB_Reset;
      A     "Lampka_pb_Stop";
      =     "DB_HMI".HMI_IN.Lampka_PB_Stop;
      A     "Lampka_pb_Cykl_Start";
      =     "DB_HMI".HMI_IN.Lampka_PB_Cykl_Start;
NETWORK
TITLE =
//Start/Stop calej lini
      A     "DB_HMI".HMI_OUT.Start_Lini_z_OP;
      =     "Blok_Para".Start_Lini_z_OP;
      A     "DB_HMI".HMI_OUT.Stop_Lini_z_OP;
      =     "Blok_Para".Stop_Lini_z_OP;
NETWORK
TITLE =
//foto_2 obrtonica to jest przod
      A(;
      O     "AIO".Obr_G15.Foto_2;
      O     "AIO".Banda_G2.Foto_2;
      );
      AN    "AIO".Obr_G15.Foto_1;
      AN    "AIO".Banda_G2.Foto_1;
      =     "M_Wypchnie_Palety";
NETWORK
TITLE = //wyjazd wtrybie auto
//Wyzwolenie wyjazdu palety gdy paleta stoi na bandzie obrotowej a nie wyjezdza
//
      A     "Zawsze_True";
      A     "DB_HMI".HMI_OUT.Wyzwolenie_Wyjazdu;
      O(;
      A     "Auto_Reczny";
      FP    "Zboczne_M44.0";
      A     "M_Wypchnie_Palety";
      A     "Blok_Para".Poz_0_st;
      AN    "M_Cykl_Bindowania_Trwa";
      );
      =     "Blok_Para".Trigger_Wyjazd;
NETWORK
TITLE = Znacznik stanu kurtyny optycznej na wlocie
//Bariery optyczne bindownicy
      AN    "AIO".Kurtyna_G25.OSSD_Tor_1_1;
      AN    "AIO".Kurtyna_G25.OSSD_Tor_1_2;
      AN    "AIO".Kurtyna_G25.OSSD_Tor_2_1;
      AN    "AIO".Kurtyna_G25.OSSD_Tor_2_2;
      =     "DB_HMI".HMI_IN.Kurtyna_Wlot_Ok;
      AN    "AIO".Kurtyna_G26.OSSD_Tor_1_1;
      AN    "AIO".Kurtyna_G26.OSSD_Tor_1_2;
      AN    "AIO".Kurtyna_G26.OSSD_Tor_2_1;
      AN    "AIO".Kurtyna_G26.OSSD_Tor_2_2;
      =     "DB_HMI".HMI_IN.Kurtyna_Wylot_Ok;
      A     "Rygiel_OK";
      =     "DB_HMI".HMI_IN.Rygiel;
NETWORK
TITLE = Znacznik pracy calej linii transportowej
      A     "Lampa_Zielona";
      =     "DB_HMI".HMI_IN.Linia_transportowa_praca;
NETWORK
TITLE = tryb pracy bindownicy: Auto(1) Reczny(0)
      A     "Blok_Bledow_Program".Blad_Krok_1;
      =     "DB_HMI".HMI_IN.Krok_1;
      A     "Blok_Bledow_Program".Blad_Krok_2;
      =     "DB_HMI".HMI_IN.Krok_2;
      A     "Blok_Bledow_Program".Blad_Krok_3;
      =     "DB_HMI".HMI_IN.Krok_3;
      A     "Blok_Bledow_Program".Blad_Krok_4;
      =     "DB_HMI".HMI_IN.Krok_4;
      A     "Blok_Bledow_Program".Blad_Krok_5;
      =     "DB_HMI".HMI_IN.Krok_5;
      A     "Blok_Bledow_Program".Blad_Krok_6;
      =     "DB_HMI".HMI_IN.Krok_6;
NETWORK
TITLE =
//przypisanie stanu wejsc i wyjsc
      L     "Bity_Przyciskow";
      T     "DB_HMI".HMI_IN.input_0;
      L     IB 1;
      T     "DB_HMI".HMI_IN.input_1;
      L     IB 2;
      T     "DB_HMI".HMI_IN.input_2;
      L     IB 3;
      T     "DB_HMI".HMI_IN.input_3;
      L     QB 0;
      T     "DB_HMI".HMI_IN.output_0;
      L     QB 1;
      T     "DB_HMI".HMI_IN.output_1;
      L     QB 2;
      T     "DB_HMI".HMI_IN.output_2;
      L     QB 3;
      T     "DB_HMI".HMI_IN.output_3;
      L     IB 8;
      T     "DB_HMI".HMI_IN.input_8;
      L     IB 9;
      T     "DB_HMI".HMI_IN.input_9;
      L     IB 10;
      T     "DB_HMI".HMI_IN.input_10;
      L     IB 11;
      T     "DB_HMI".HMI_IN.input_11;
NETWORK
TITLE = krok 1 trybu pracy
//Przypisanie aktualnych krokow 
//krok_1  - jedz na pozycje 
      A     "Blok_Para".Krok_1;
      L     1;
      JC    tr;
//krok_2 - szukaj srodka 
      A     "Blok_Para".krok_2;
      L     2;
      JC    tr;
//krok_3 - jedz na prawo
      A     "Blok_Para".krok_3;
      L     3;
      JC    tr;
//krok_4 - strzelaj 
      A     "Blok_Para".krok_4;
      L     4;
      JC    tr;
//krok_5  - pauza po strzale
      A     "Blok_Para".krok_5;
      L     5;
      JC    tr;
//krok_6 - jedz do srodka
      A     "Blok_Para".krok_6;
      L     6;
      JC    tr;
//daj 0
      L     0;
tr:   T     "DB_HMI".HMI_IN.INT_Liczba_Akt_Kroku;
NETWORK
TITLE = znacznik migania bledu
//Sprawdzenie czy sa bledy jak sa to miganie bledow
      SET;
      R     "DB_HMI".HMI_IN.Znacznik_Migania_Bledu;
      O(;
      L     DB119.DBD 0;
      L     0;
      <>D;
      );
      O(;
      L     DB119.DBD 4;
      L     0;
      <>D;
      );
      O(;
      L     DB119.DBD 8;
      L     0;
      <>D;
      );
      S     "DB_HMI".HMI_IN.Znacznik_Migania_Bledu;
NETWORK
TITLE = czujnik prasy s 22
//Obsluga wygladu prasy
//
      A     "Prasa_W_Gorze";
      =     "DB_HMI".HMI_IN.Czujnik_Prasa;
//zawor prasa
      AN    "Zawor_Prasa";
      =     "DB_HMI".HMI_IN.Stan_Zaworu;
NETWORK
TITLE =
//Aktualizacja godziny/daty panela z godzina/czasem PLC
      CALL  "READ_CLK" (
           RET_VAL                  := #LW0_Help,
           CDT                      := "DB_HMI".HMI_IN.Aktualna_Data);
NETWORK
TITLE =
//Obrotnica na Genderze
//
      A(;
      O     "AIO".Czuj_G19_B.Czujnik_0_St;
      O     "AIO".Czuj_G17_B.Czujnik_180_St;
      );
      R     DB120.DBX 13.0;
      A(;
      O     "AIO".Czuj_G19_B.Czujnik_90_St;
      O     "AIO".Czuj_G17_B.Czujnik_270_St;
      );
      S     DB120.DBX 13.0;
      A     DB120.DBX 13.0;
      =     "DB_HMI".HMI_IN.Obr_Gender_Wzdluz;
NETWORK
TITLE =
//obrotnica za Genderem
      AN    "AIO".Czuj_T19.Czujnik_90_St;
      =     L 2.0;
      A     L 2.0;
      BLD   102;
      =     "DB_HMI".HMI_IN.Obr_za_Genderem_wzdluz;
      A     L 2.0;
      S     DB120.DBX 14.0;
      A     "AIO".Czuj_T19.Czujnik_90_St;
      R     DB120.DBX 14.0;
      NOP   0;
NETWORK
TITLE =
//Obrotnica za foliarka
      A     "AIO".Czuj_T21.Czujnik_0_St;
      =     L 2.0;
      A     L 2.0;
      BLD   102;
      =     "DB_HMI".HMI_IN.Obr_za_Foliarka_wzdluz;
      A     L 2.0;
      S     DB120.DBX 15.0;
      A     "AIO".Czuj_T21.Czujnik_90_St;
      R     DB120.DBX 15.0;
      NOP   0;
NETWORK
TITLE =
      A     DB310.DBX 0.7;
      =     L 2.0;
      A     L 2.0;
      JNB   _001;
      L     "Rejestr Band".Tasma_Wozek_0;
      T     "Rejestr_Band_HMI".Tasma_Wozek_0_HMI;
_001: NOP   0;
      A     L 2.0;
      NOT;
      JNB   _002;
      L     0;
      T     "Rejestr_Band_HMI".Tasma_Wozek_0_HMI;
_002: NOP   0;
NETWORK
TITLE =
      A     DB310.DBX 4.7;
      =     L 2.0;
      A     L 2.0;
      JNB   _003;
      L     "Rejestr Band".Tasma_Gender_1;
      T     "Rejestr_Band_HMI".Tasma_Gender_1_HMI;
_003: NOP   0;
      A     L 2.0;
      NOT;
      JNB   _004;
      L     0;
      T     "Rejestr_Band_HMI".Tasma_Gender_1_HMI;
_004: NOP   0;
NETWORK
TITLE =
      A     DB310.DBX 8.7;
      =     L 2.0;
      A     L 2.0;
      JNB   _005;
      L     "Rejestr Band".Tasma_Gender_2;
      T     "Rejestr_Band_HMI".Tasma_Gender_2_HMI;
_005: NOP   0;
      A     L 2.0;
      NOT;
      JNB   _006;
      L     0;
      T     "Rejestr_Band_HMI".Tasma_Gender_2_HMI;
_006: NOP   0;
NETWORK
TITLE =
      A     DB310.DBX 12.7;
      =     L 2.0;
      A     L 2.0;
      JNB   _007;
      L     "Rejestr Band".Tasma_Gender_Obr_3;
      T     "Rejestr_Band_HMI".Tasma_Gender_Obr_3_HMI;
_007: NOP   0;
      A     L 2.0;
      NOT;
      JNB   _008;
      L     0;
      T     "Rejestr_Band_HMI".Tasma_Gender_Obr_3_HMI;
_008: NOP   0;
NETWORK
TITLE =
      A     DB310.DBX 16.7;
      =     L 2.0;
      A     L 2.0;
      JNB   _009;
      L     "Rejestr Band".Tasma_Gender_4;
      T     "Rejestr_Band_HMI".Tasma_Gender_4_HMI;
_009: NOP   0;
      A     L 2.0;
      NOT;
      JNB   _00a;
      L     0;
      T     "Rejestr_Band_HMI".Tasma_Gender_4_HMI;
_00a: NOP   0;
NETWORK
TITLE =
      A     DB310.DBX 20.7;
      =     L 2.0;
      A     L 2.0;
      JNB   _00b;
      L     "Rejestr Band".Tasma_Transp_Obr_4;
      T     "Rejestr_Band_HMI".Tasma_Transp_Obr_4_HMI;
_00b: NOP   0;
      A     L 2.0;
      NOT;
      JNB   _00c;
      L     0;
      T     "Rejestr_Band_HMI".Tasma_Transp_Obr_4_HMI;
_00c: NOP   0;
NETWORK
TITLE =
      A     DB310.DBX 24.7;
      =     L 2.0;
      A     L 2.0;
      JNB   _00d;
      L     "Rejestr Band".Tasma_Transp_3;
      T     "Rejestr_Band_HMI".Tasma_Transp_3_HMI;
_00d: NOP   0;
      A     L 2.0;
      NOT;
      JNB   _00e;
      L     0;
      T     "Rejestr_Band_HMI".Tasma_Transp_3_HMI;
_00e: NOP   0;
NETWORK
TITLE =
      A     DB310.DBX 28.7;
      =     L 2.0;
      A     L 2.0;
      JNB   _00f;
      L     "Rejestr Band".Tasma_Transp_5;
      T     "Rejestr_Band_HMI".Tasma_Transp_5_HMI;
_00f: NOP   0;
      A     L 2.0;
      NOT;
      JNB   _010;
      L     0;
      T     "Rejestr_Band_HMI".Tasma_Transp_5_HMI;
_010: NOP   0;
NETWORK
TITLE =
      A     DB310.DBX 32.7;
      =     L 2.0;
      A     L 2.0;
      JNB   _011;
      L     "Rejestr Band".Tasma_Transp_6;
      T     "Rejestr_Band_HMI".Tasma_Transp_6_HMI;
_011: NOP   0;
      A     L 2.0;
      NOT;
      JNB   _012;
      L     0;
      T     "Rejestr_Band_HMI".Tasma_Transp_6_HMI;
_012: NOP   0;
NETWORK
TITLE =
      A     DB310.DBX 36.7;
      =     L 2.0;
      A     L 2.0;
      JNB   _013;
      L     "Rejestr Band".Tasma_Transp_7;
      T     "Rejestr_Band_HMI".Tasma_Transp_7_HMI;
_013: NOP   0;
      A     L 2.0;
      NOT;
      JNB   _014;
      L     0;
      T     "Rejestr_Band_HMI".Tasma_Transp_7_HMI;
_014: NOP   0;
NETWORK
TITLE =
      A     DB310.DBX 40.7;
      =     L 2.0;
      A     L 2.0;
      JNB   _015;
      L     "Rejestr Band".Tasma_Transp_8;
      T     "Rejestr_Band_HMI".Tasma_Transp_8_HMI;
_015: NOP   0;
      A     L 2.0;
      NOT;
      JNB   _016;
      L     0;
      T     "Rejestr_Band_HMI".Tasma_Transp_8_HMI;
_016: NOP   0;
NETWORK
TITLE =
      A     DB310.DBX 44.7;
      =     L 2.0;
      A     L 2.0;
      JNB   _017;
      L     "Rejestr Band".Tasma_Transp_9;
      T     "Rejestr_Band_HMI".Tasma_Transp_9_HMI;
_017: NOP   0;
      A     L 2.0;
      NOT;
      JNB   _018;
      L     0;
      T     "Rejestr_Band_HMI".Tasma_Transp_9_HMI;
_018: NOP   0;
NETWORK
TITLE =
      A     DB310.DBX 48.7;
      =     L 2.0;
      A     L 2.0;
      JNB   _019;
      L     "Rejestr Band".Tasma_Transp_10_Fol;
      T     "Rejestr_Band_HMI".Tasma_Transp_10_Fol_HMI;
_019: NOP   0;
      A     L 2.0;
      NOT;
      JNB   _01a;
      L     0;
      T     "Rejestr_Band_HMI".Tasma_Transp_10_Fol_HMI;
_01a: NOP   0;
NETWORK
TITLE =
      A     DB310.DBX 52.7;
      =     L 2.0;
      A     L 2.0;
      JNB   _01b;
      L     "Rejestr Band".Tasma_Transp_4_Fol;
      T     "Rejestr_Band_HMI".Tasma_Transp_4_Fol_HMI;
_01b: NOP   0;
      A     L 2.0;
      NOT;
      JNB   _01c;
      L     0;
      T     "Rejestr_Band_HMI".Tasma_Transp_4_Fol_HMI;
_01c: NOP   0;
NETWORK
TITLE =
      A     DB310.DBX 56.7;
      =     L 2.0;
      A     L 2.0;
      JNB   _01d;
      L     "Rejestr Band".Tasma_Transp_Obr_Fol;
      T     "Rejestr_Band_HMI".Tasma_Transp_Obr_Fol_HMI;
_01d: NOP   0;
      A     L 2.0;
      NOT;
      JNB   _01e;
      L     0;
      T     "Rejestr_Band_HMI".Tasma_Transp_Obr_Fol_HMI;
_01e: NOP   0;
NETWORK
TITLE =
      A     DB310.DBX 60.7;
      =     L 2.0;
      A     L 2.0;
      JNB   _01f;
      L     "Rejestr Band".Tasma_Transp_6_Fol;
      T     "Rejestr_Band_HMI".Tasma_Transp_6_Fol_HMI;
_01f: NOP   0;
      A     L 2.0;
      NOT;
      JNB   _020;
      L     0;
      T     "Rejestr_Band_HMI".Tasma_Transp_6_Fol_HMI;
_020: NOP   0;
NETWORK
TITLE =
      A     DB310.DBX 64.7;
      =     L 2.0;
      A     L 2.0;
      JNB   _021;
      L     "Rejestr Band".Tasma_Transp_11_Fol;
      T     "Rejestr_Band_HMI".Tasma_Transp_11_Fol_HMI;
_021: NOP   0;
      A     L 2.0;
      NOT;
      JNB   _022;
      L     0;
      T     "Rejestr_Band_HMI".Tasma_Transp_11_Fol_HMI;
_022: NOP   0;
NETWORK
TITLE =
      A     DB310.DBX 68.7;
      =     L 2.0;
      A     L 2.0;
      JNB   _023;
      L     "Rejestr Band".Tasma_Transp_12;
      T     "Rejestr_Band_HMI".Tasma_Transp_12_HMI;
_023: NOP   0;
      A     L 2.0;
      NOT;
      JNB   _024;
      L     0;
      T     "Rejestr_Band_HMI".Tasma_Transp_12_HMI;
_024: NOP   0;
NETWORK
TITLE =
      A     DB310.DBX 72.7;
      =     L 2.0;
      A     L 2.0;
      JNB   _025;
      L     "Rejestr Band".Tasma_Transp_Obr_13;
      T     "Rejestr_Band_HMI".Tasma_Transp_Obr_13_HMI;
_025: NOP   0;
      A     L 2.0;
      NOT;
      JNB   _026;
      L     0;
      T     "Rejestr_Band_HMI".Tasma_Transp_Obr_13_HMI;
_026: NOP   0;
NETWORK
TITLE =
      A     DB310.DBX 76.7;
      =     L 2.0;
      A     L 2.0;
      JNB   _027;
      L     "Rejestr Band".Tasma_Wysjsciowa_14;
      T     "Rejestr_Band_HMI".Tasma_Wysjsciowa_14_HMI;
_027: NOP   0;
      A     L 2.0;
      NOT;
      JNB   _028;
      L     0;
      T     "Rejestr_Band_HMI".Tasma_Wysjsciowa_14_HMI;
_028: NOP   0;
END_FUNCTION

FUNCTION "Funkcja_Zegara" : VOID	// FC 140
AUTHOR : Kng
NAME : HELP_FC
VERSION : 0.1
VAR_INPUT
  Timer_NR : TIMER ;
  Czas : S5TIME ;
END_VAR
VAR_IN_OUT
  Wyjscie : BOOL ;
END_VAR
BEGIN
NETWORK
TITLE =
      A     #Timer_NR;
      SAVE;
      NOT;
      L     #Czas;
      SD    #Timer_NR;
      X     BR;
      X     #Wyjscie;
      =     #Wyjscie;
END_FUNCTION

FUNCTION "Komunikacja_Gender" : VOID	// FC 205
//Marki 400. Bity sa widziane od strony odbierania
VERSION : 0.1
BEGIN
NETWORK
TITLE =
//Ten Network celowo jest wolny
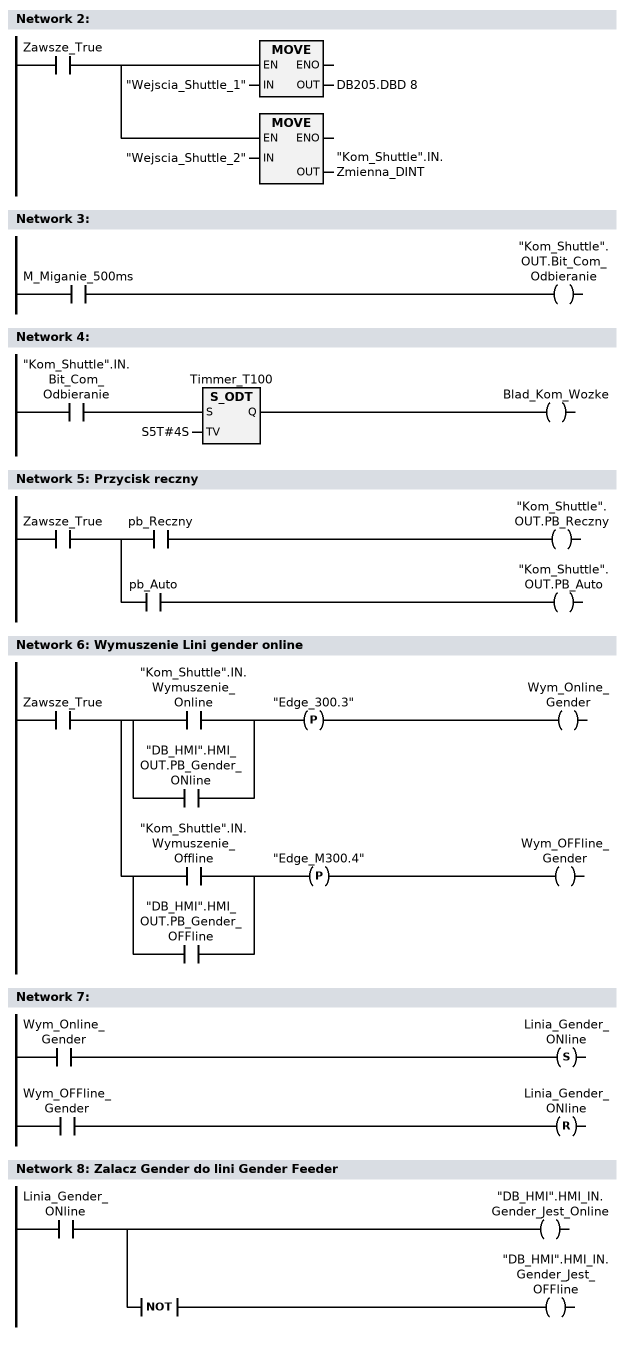
NETWORK
TITLE =
//Przypisanie danych z dp coupler
      A     "Zawsze_True";
      =     L 0.0;
      A     L 0.0;
      JNB   _001;
      L     "Wejscia_Shuttle_1";
      T     DB205.DBD 8;
_001: NOP   0;
      A     L 0.0;
      JNB   _002;
      L     "Wejscia_Shuttle_2";
      T     "Kom_Shuttle".IN.Zmienna_DINT;
_002: NOP   0;
NETWORK
TITLE =
//Komunikacj z Gender
      A     "M_Miganie_500ms";
      =     "Kom_Shuttle".OUT.Bit_Com_Odbieranie;
NETWORK
TITLE =
//Sprawdzenie czy komunikacja jest OK
      A     "Kom_Shuttle".IN.Bit_Com_Odbieranie;
      L     S5T#4S;
      SD    "Timmer_T100";
      NOP   0;
      NOP   0;
      NOP   0;
      A     "Timmer_T100";
      =     "Blad_Kom_Wozke";
NETWORK
TITLE = Przycisk reczny
//Przycisk reczny
      A     "Zawsze_True";
      =     L 0.0;
      A     L 0.0;
      A     "pb_Reczny";
      =     "Kom_Shuttle".OUT.PB_Reczny;
      A     L 0.0;
      A     "pb_Auto";
      =     "Kom_Shuttle".OUT.PB_Auto;
NETWORK
TITLE = Wymuszenie Lini gender online
//Wymus online/offline
      A     "Zawsze_True";
      =     L 0.0;
      A     L 0.0;
      A(;
      O     "Kom_Shuttle".IN.Wymuszenie_Online;
      O     "DB_HMI".HMI_OUT.PB_Gender_ONline;
      );
      FP    "Edge_300.3";
      =     "Wym_Online_Gender";
      A     L 0.0;
      A(;
      O     "Kom_Shuttle".IN.Wymuszenie_Offline;
      O     "DB_HMI".HMI_OUT.PB_Gender_OFFline;
      );
      FP    "Edge_M300.4";
      =     "Wym_OFFline_Gender";
NETWORK
TITLE =
//Wymuszenie Lini Gender online /offline
      A     "Wym_Online_Gender";
      S     "Linia_Gender_ONline";
      A     "Wym_OFFline_Gender";
      R     "Linia_Gender_ONline";
      NOP   0;
NETWORK
TITLE = Zalacz Gender do lini Gender Feeder
//Sprawdzenie czy Gender jest offline czy online
      A     "Linia_Gender_ONline";
      =     L 0.0;
      A     L 0.0;
      BLD   102;
      =     "DB_HMI".HMI_IN.Gender_Jest_Online;
      A     L 0.0;
      NOT;
      =     "DB_HMI".HMI_IN.Gender_Jest_OFFline;
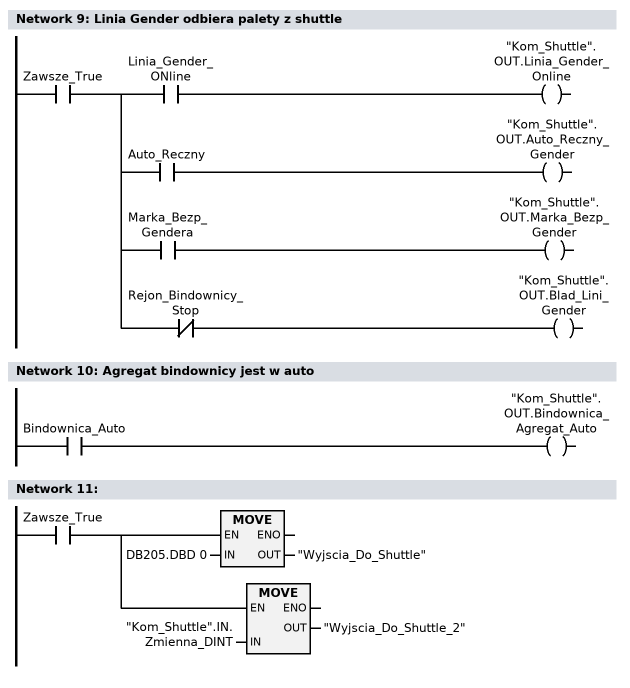
NETWORK
TITLE = Linia Gender odbiera palety z shuttle
//Wyswietlenie stanu pracy
      A     "Zawsze_True";
      =     L 0.0;
      A     L 0.0;
      A     "Linia_Gender_ONline";
      =     "Kom_Shuttle".OUT.Linia_Gender_Online;
      A     L 0.0;
      A     "Auto_Reczny";
      =     "Kom_Shuttle".OUT.Auto_Reczny_Gender;
      A     L 0.0;
      A     "Marka_Bezp_Gendera";
      =     "Kom_Shuttle".OUT.Marka_Bezp_Gender;
      A     L 0.0;
      AN    "Rejon_Bindownicy_Stop";
      =     "Kom_Shuttle".OUT.Blad_Lini_Gender;
NETWORK
TITLE = Agregat bindownicy jest w auto
      A     "Bindownica_Auto";
      =     "Kom_Shuttle".OUT.Bindownica_Agregat_Auto;
NETWORK
TITLE =
//Przypisanie danych z dp coupler
      A     "Zawsze_True";
      =     L 0.0;
      A     L 0.0;
      JNB   _003;
      L     DB205.DBD 0;
      T     "Wyjscia_Do_Shuttle";
_003: NOP   0;
      A     L 0.0;
      JNB   _004;
      L     "Kom_Shuttle".IN.Zmienna_DINT;
      T     "Wyjscia_Do_Shuttle_2";
_004: NOP   0;
END_FUNCTION

FUNCTION "Monitor_Band_Lini" : VOID	// FC 310
//Funkcja monitoru band dla transportera
//
//Bajty m600
//Foto 1 to foto przod
//foto 2 to foto tyl 
//wyjatek to obrotnica :
//gdzye foto 1 -tyl
//foto 2- przod
AUTHOR : Kng
NAME : Main
VERSION : 0.1
VAR_TEMP
  Temp_Bit_1 : BOOL ;
  Temp_Bit_2 : BOOL ;
END_VAR
BEGIN
NETWORK
TITLE =
//Ten network celowo jest wolny
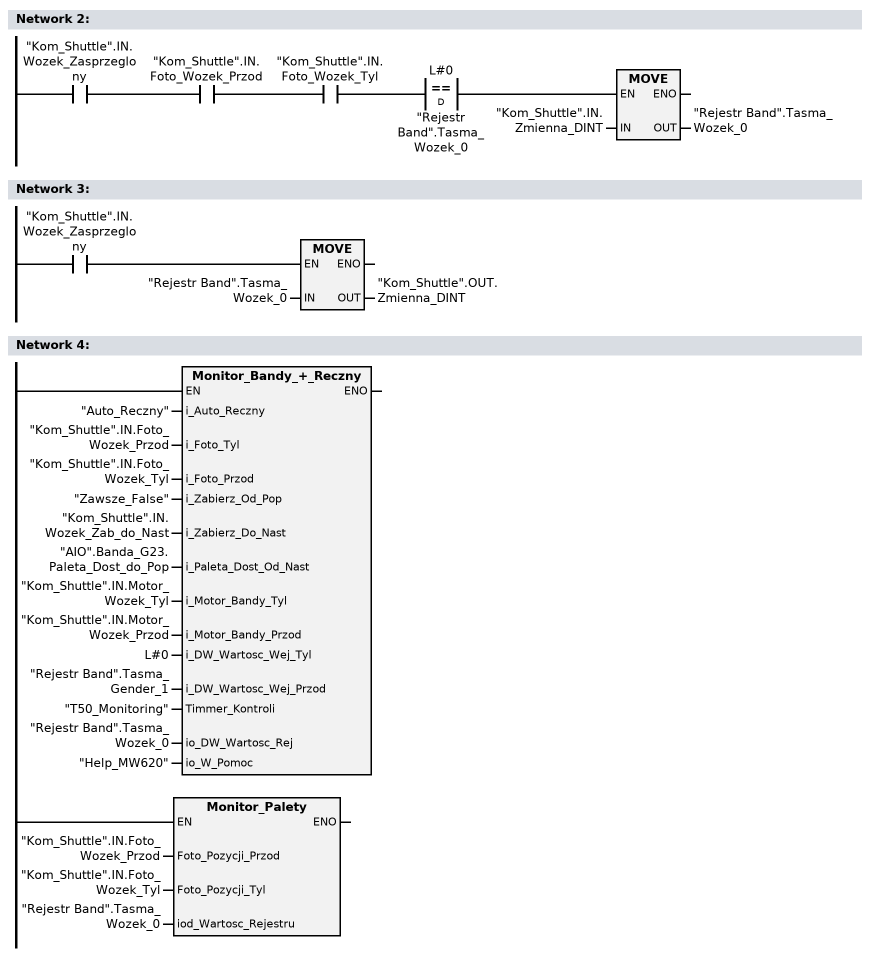
NETWORK
TITLE =
      A     "Kom_Shuttle".IN.Wozek_Zasprzeglony;
      A     "Kom_Shuttle".IN.Foto_Wozek_Przod;
      A     "Kom_Shuttle".IN.Foto_Wozek_Tyl;
      A(;
      L     L#0;
      L     "Rejestr Band".Tasma_Wozek_0;
      ==D;
      );
      JNB   _001;
      L     "Kom_Shuttle".IN.Zmienna_DINT;
      T     "Rejestr Band".Tasma_Wozek_0;
_001: NOP   0;
NETWORK
TITLE =
//Przepisanie wartosc do wozka
      A     "Kom_Shuttle".IN.Wozek_Zasprzeglony;
      JNB   _002;
      L     "Rejestr Band".Tasma_Wozek_0;
      T     "Kom_Shuttle".OUT.Zmienna_DINT;
_002: NOP   0;
NETWORK
TITLE =
//Banda zerowa to banda wozek
      CALL  "Monitor_Bandy_+_Reczny" (
           i_Auto_Reczny            := "Auto_Reczny",
           i_Foto_Tyl               := "Kom_Shuttle".IN.Foto_Wozek_Przod,
           i_Foto_Przod             := "Kom_Shuttle".IN.Foto_Wozek_Tyl,
           i_Zabierz_Od_Pop         := "Zawsze_False",
           i_Zabierz_Do_Nast        := "Kom_Shuttle".IN.Wozek_Zab_do_Nast,
           i_Paleta_Dost_Od_Nast    := "AIO".Banda_G23.Paleta_Dost_do_Pop,
           i_Motor_Bandy_Tyl        := "Kom_Shuttle".IN.Motor_Wozek_Tyl,
           i_Motor_Bandy_Przod      := "Kom_Shuttle".IN.Motor_Wozek_Przod,
           i_DW_Wartosc_Wej_Tyl     := L#0,
           i_DW_Wartosc_Wej_Przod   := "Rejestr Band".Tasma_Gender_1,
           Timmer_Kontroli          := "T50_Monitoring",
           io_DW_Wartosc_Rej        := "Rejestr Band".Tasma_Wozek_0,
           io_W_Pomoc               := "Help_MW620");
//Monitor palety
      CALL  "Monitor_Palety" (
           Foto_Pozycji_Przod       := "Kom_Shuttle".IN.Foto_Wozek_Przod,
           Foto_Pozycji_Tyl         := "Kom_Shuttle".IN.Foto_Wozek_Tyl,
           iod_Wartosc_Rejestru     := "Rejestr Band".Tasma_Wozek_0);
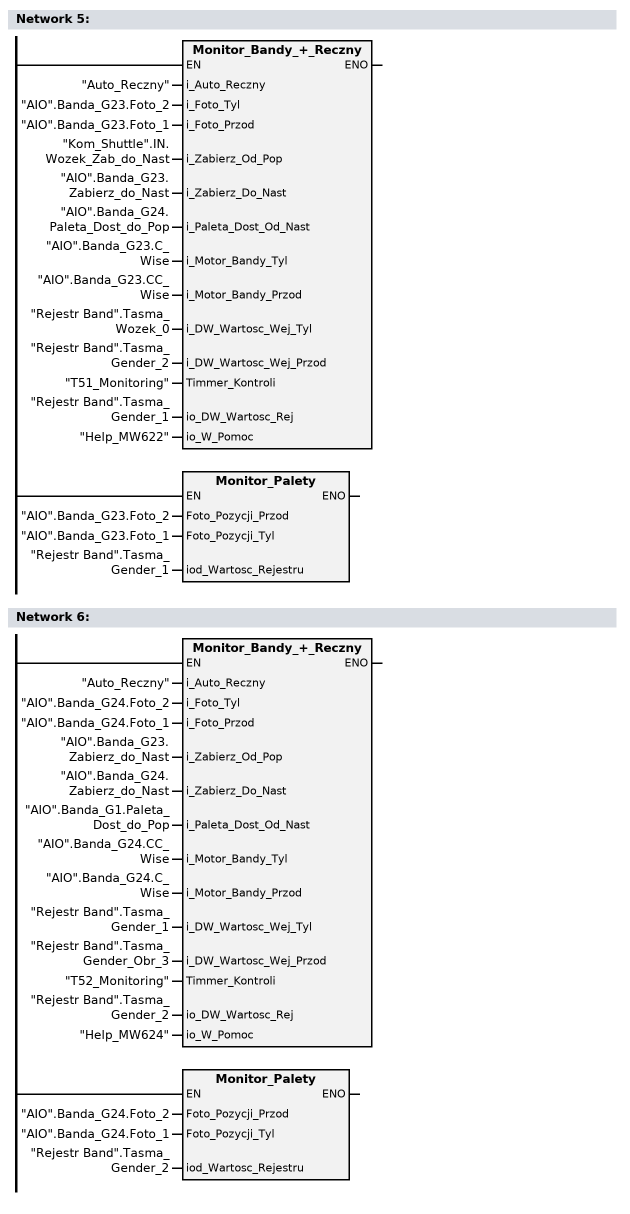
NETWORK
TITLE =
//Banda pierwsza to gender tasma 1 
//Foto 1 to foto przod
//foto 2 to foto tyl 
//wyjatek to obrotnica :
//gdzye foto 1 -tyl
//foto 2- przod
      CALL  "Monitor_Bandy_+_Reczny" (
           i_Auto_Reczny            := "Auto_Reczny",
           i_Foto_Tyl               := "AIO".Banda_G23.Foto_2,
           i_Foto_Przod             := "AIO".Banda_G23.Foto_1,
           i_Zabierz_Od_Pop         := "Kom_Shuttle".IN.Wozek_Zab_do_Nast,
           i_Zabierz_Do_Nast        := "AIO".Banda_G23.Zabierz_do_Nast,
           i_Paleta_Dost_Od_Nast    := "AIO".Banda_G24.Paleta_Dost_do_Pop,
           i_Motor_Bandy_Tyl        := "AIO".Banda_G23.C_Wise,
           i_Motor_Bandy_Przod      := "AIO".Banda_G23.CC_Wise,
           i_DW_Wartosc_Wej_Tyl     := "Rejestr Band".Tasma_Wozek_0,
           i_DW_Wartosc_Wej_Przod   := "Rejestr Band".Tasma_Gender_2,
           Timmer_Kontroli          := "T51_Monitoring",
           io_DW_Wartosc_Rej        := "Rejestr Band".Tasma_Gender_1,
           io_W_Pomoc               := "Help_MW622");
      CALL  "Monitor_Palety" (
           Foto_Pozycji_Przod       := "AIO".Banda_G23.Foto_2,
           Foto_Pozycji_Tyl         := "AIO".Banda_G23.Foto_1,
           iod_Wartosc_Rejestru     := "Rejestr Band".Tasma_Gender_1);
NETWORK
TITLE =
//Tasma 2 Gender w adresacji 24
      CALL  "Monitor_Bandy_+_Reczny" (
           i_Auto_Reczny            := "Auto_Reczny",
           i_Foto_Tyl               := "AIO".Banda_G24.Foto_2,
           i_Foto_Przod             := "AIO".Banda_G24.Foto_1,
           i_Zabierz_Od_Pop         := "AIO".Banda_G23.Zabierz_do_Nast,
           i_Zabierz_Do_Nast        := "AIO".Banda_G24.Zabierz_do_Nast,
           i_Paleta_Dost_Od_Nast    := "AIO".Banda_G1.Paleta_Dost_do_Pop,
           i_Motor_Bandy_Tyl        := "AIO".Banda_G24.CC_Wise,
           i_Motor_Bandy_Przod      := "AIO".Banda_G24.C_Wise,
           i_DW_Wartosc_Wej_Tyl     := "Rejestr Band".Tasma_Gender_1,
           i_DW_Wartosc_Wej_Przod   := "Rejestr Band".Tasma_Gender_Obr_3,
           Timmer_Kontroli          := "T52_Monitoring",
           io_DW_Wartosc_Rej        := "Rejestr Band".Tasma_Gender_2,
           io_W_Pomoc               := "Help_MW624");
      CALL  "Monitor_Palety" (
           Foto_Pozycji_Przod       := "AIO".Banda_G24.Foto_2,
           Foto_Pozycji_Tyl         := "AIO".Banda_G24.Foto_1,
           iod_Wartosc_Rejestru     := "Rejestr Band".Tasma_Gender_2);
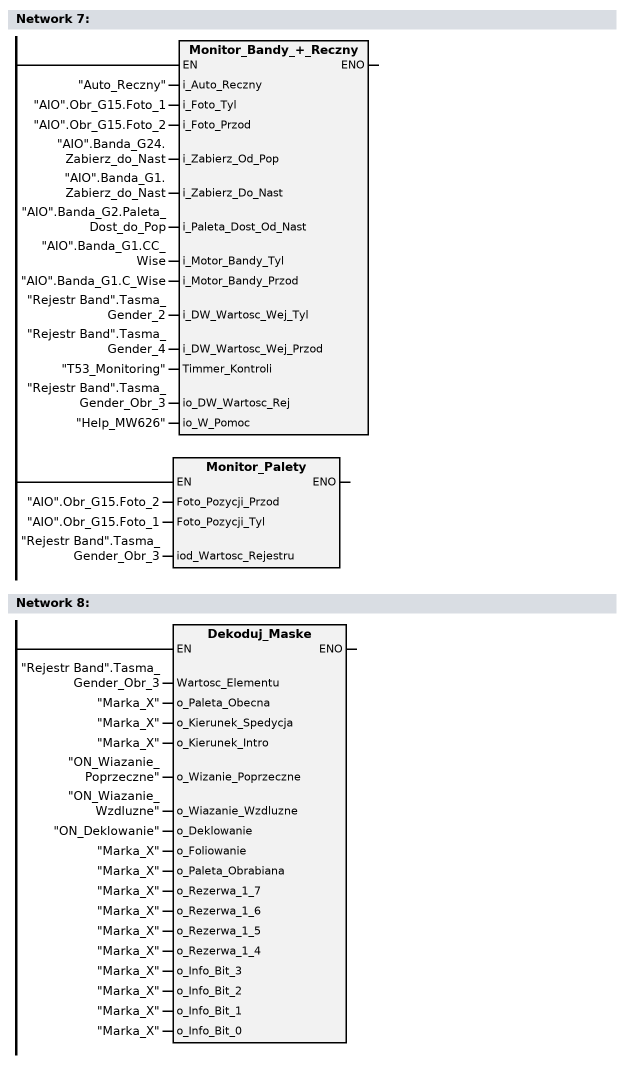
NETWORK
TITLE =
//Tasma Obrotnica o adresie 1
      CALL  "Monitor_Bandy_+_Reczny" (
           i_Auto_Reczny            := "Auto_Reczny",
           i_Foto_Tyl               := "AIO".Obr_G15.Foto_1,
           i_Foto_Przod             := "AIO".Obr_G15.Foto_2,
           i_Zabierz_Od_Pop         := "AIO".Banda_G24.Zabierz_do_Nast,
           i_Zabierz_Do_Nast        := "AIO".Banda_G1.Zabierz_do_Nast,
           i_Paleta_Dost_Od_Nast    := "AIO".Banda_G2.Paleta_Dost_do_Pop,
           i_Motor_Bandy_Tyl        := "AIO".Banda_G1.CC_Wise,
           i_Motor_Bandy_Przod      := "AIO".Banda_G1.C_Wise,
           i_DW_Wartosc_Wej_Tyl     := "Rejestr Band".Tasma_Gender_2,
           i_DW_Wartosc_Wej_Przod   := "Rejestr Band".Tasma_Gender_4,
           Timmer_Kontroli          := "T53_Monitoring",
           io_DW_Wartosc_Rej        := "Rejestr Band".Tasma_Gender_Obr_3,
           io_W_Pomoc               := "Help_MW626");
      CALL  "Monitor_Palety" (
           Foto_Pozycji_Przod       := "AIO".Obr_G15.Foto_2,
           Foto_Pozycji_Tyl         := "AIO".Obr_G15.Foto_1,
           iod_Wartosc_Rejestru     := "Rejestr Band".Tasma_Gender_Obr_3);
NETWORK
TITLE =
//Dekodowanie maski. Aby umozliwic bindowanie
//-Obsluga wiazan jest w FC120
//-Obsluga Dekla jest w FB3
//
      CALL  "Dekoduj_Maske" (
           Wartosc_Elementu         := "Rejestr Band".Tasma_Gender_Obr_3,
           o_Paleta_Obecna          := "Marka_X",
           o_Kierunek_Spedycja      := "Marka_X",
           o_Kierunek_Intro         := "Marka_X",
           o_Wizanie_Poprzeczne     := "ON_Wiazanie_Poprzeczne",
           o_Wiazanie_Wzdluzne      := "ON_Wiazanie_Wzdluzne",
           o_Deklowanie             := "ON_Deklowanie",
           o_Foliowanie             := "Marka_X",
           o_Paleta_Obrabiana       := "Marka_X",
           o_Rezerwa_1_7            := "Marka_X",
           o_Rezerwa_1_6            := "Marka_X",
           o_Rezerwa_1_5            := "Marka_X",
           o_Rezerwa_1_4            := "Marka_X",
           o_Info_Bit_3             := "Marka_X",
           o_Info_Bit_2             := "Marka_X",
           o_Info_Bit_1             := "Marka_X",
           o_Info_Bit_0             := "Marka_X");
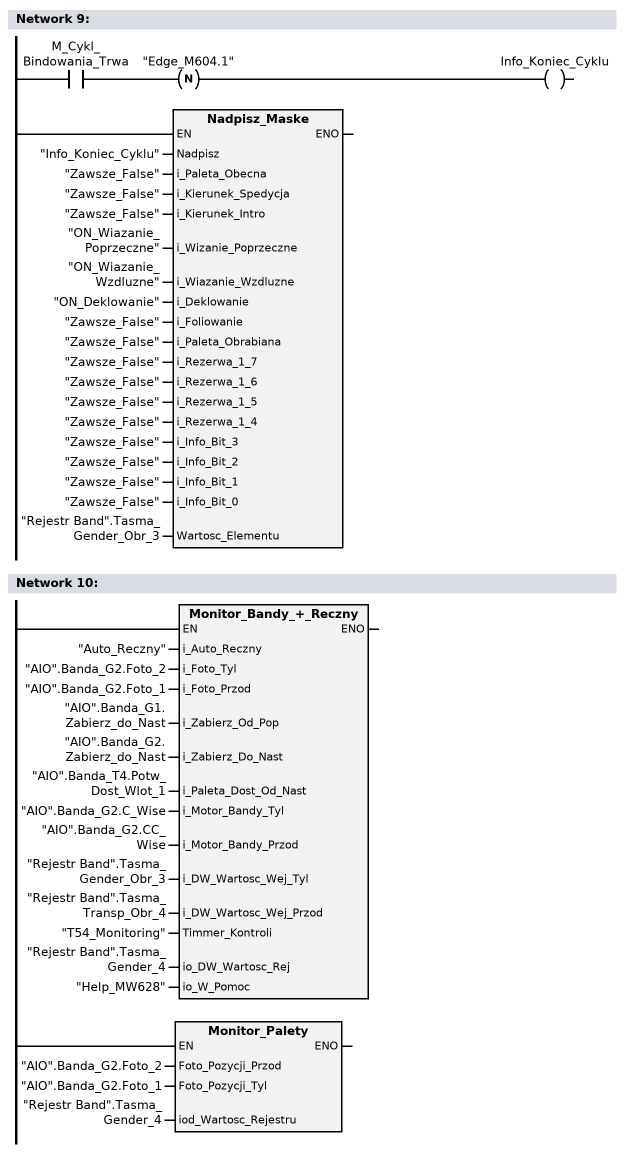
NETWORK
TITLE =
//Nadpisz Maske
      A     "M_Cykl_Bindowania_Trwa";
      FN    "Edge_M604.1";
      =     "Info_Koniec_Cyklu";
      CALL  "Nadpisz_Maske" (
           Nadpisz                  := "Info_Koniec_Cyklu",
           i_Paleta_Obecna          := "Zawsze_False",
           i_Kierunek_Spedycja      := "Zawsze_False",
           i_Kierunek_Intro         := "Zawsze_False",
           i_Wizanie_Poprzeczne     := "ON_Wiazanie_Poprzeczne",
           i_Wiazanie_Wzdluzne      := "ON_Wiazanie_Wzdluzne",
           i_Deklowanie             := "ON_Deklowanie",
           i_Foliowanie             := "Zawsze_False",
           i_Paleta_Obrabiana       := "Zawsze_False",
           i_Rezerwa_1_7            := "Zawsze_False",
           i_Rezerwa_1_6            := "Zawsze_False",
           i_Rezerwa_1_5            := "Zawsze_False",
           i_Rezerwa_1_4            := "Zawsze_False",
           i_Info_Bit_3             := "Zawsze_False",
           i_Info_Bit_2             := "Zawsze_False",
           i_Info_Bit_1             := "Zawsze_False",
           i_Info_Bit_0             := "Zawsze_False",
           Wartosc_Elementu         := "Rejestr Band".Tasma_Gender_Obr_3);
NETWORK
TITLE =
//Tasma 4 Ostatnia Gender 
      CALL  "Monitor_Bandy_+_Reczny" (
           i_Auto_Reczny            := "Auto_Reczny",
           i_Foto_Tyl               := "AIO".Banda_G2.Foto_2,
           i_Foto_Przod             := "AIO".Banda_G2.Foto_1,
           i_Zabierz_Od_Pop         := "AIO".Banda_G1.Zabierz_do_Nast,
           i_Zabierz_Do_Nast        := "AIO".Banda_G2.Zabierz_do_Nast,
           i_Paleta_Dost_Od_Nast    := "AIO".Banda_T4.Potw_Dost_Wlot_1,
           i_Motor_Bandy_Tyl        := "AIO".Banda_G2.C_Wise,
           i_Motor_Bandy_Przod      := "AIO".Banda_G2.CC_Wise,
           i_DW_Wartosc_Wej_Tyl     := "Rejestr Band".Tasma_Gender_Obr_3,
           i_DW_Wartosc_Wej_Przod   := "Rejestr Band".Tasma_Transp_Obr_4,
           Timmer_Kontroli          := "T54_Monitoring",
           io_DW_Wartosc_Rej        := "Rejestr Band".Tasma_Gender_4,
           io_W_Pomoc               := "Help_MW628");
      CALL  "Monitor_Palety" (
           Foto_Pozycji_Przod       := "AIO".Banda_G2.Foto_2,
           Foto_Pozycji_Tyl         := "AIO".Banda_G2.Foto_1,
           iod_Wartosc_Rejestru     := "Rejestr Band".Tasma_Gender_4);
